// TIA Portal V21 program export: 0 tag tables, 0 data types, 1 data blocks, 5 code blocks (in call order from the OBs), 1 instance data blocks

DATA_BLOCK "Calc"   // DB1
{ S7_Optimized_Access := 'TRUE' }
// stored: MemoryReserve 100
   VAR
      reale : Array[0..100] of LReal;
      tempociclo : LReal;
      tempociclo_T : LReal;
      interi : Array[0..10] of Int;
      tempo : LReal;
      pulse : Array[0..30] of Bool;
   END_VAR
BEGIN
END_DATA_BLOCK

ORGANIZATION_BLOCK "Main"   // OB1, LAD, ProgramCycle
TITLE = "Main Program Sweep (Cycle)"
{ S7_Optimized_Access := 'TRUE' }
// stored: SetENOAutomatically false
   VAR_INPUT
      Initial_Call : Bool;
      Remanence : Bool;
   END_VAR
   VAR_TEMP
      virposINT : DInt;
   END_VAR
BEGIN
END_ORGANIZATION_BLOCK

ORGANIZATION_BLOCK "Cyclic interrupt"   // OB30, LAD, CyclicInterrupt
{ S7_Optimized_Access := 'TRUE' }
// stored: CyclicTime 5000, SetENOAutomatically false
   VAR_INPUT
      Initial_Call : Bool;
      Event_Count : Int;
   END_VAR
   VAR_TEMP
      virposINT : DInt;
      appo : Real;
      VirOnTarget : Bool;
   END_VAR
   VAR_TEMP   // added for the SCL form of the ladder/FBD networks
      _w1 : Bool;
      _w2 : Bool;
      _w3 : Bool;
      _w4 : Bool;
      _w5 : Bool;
      _w6 : Bool;
   END_VAR
BEGIN

REGION Network 2
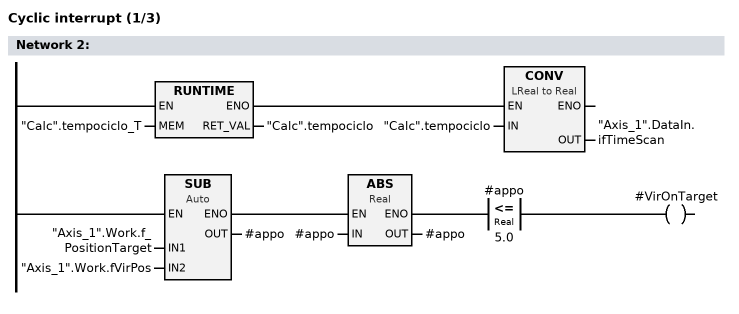
   // no SCL statement known for Runtime: written as a call
   // ENO of a box is taken as its EN; it also drops when the box reports an error
   "Calc".tempociclo := Runtime(mem := "Calc".tempociclo_T);
   "Axis_1".DataIn.ifTimeScan := LREAL_TO_REAL("Calc".tempociclo);
   #appo := "Axis_1".Work.f_PositionTarget - "Axis_1".Work.fVirPos;
   #appo := ABS(#appo);
   #VirOnTarget := #appo <= 5.0;
END_REGION

REGION Network 3
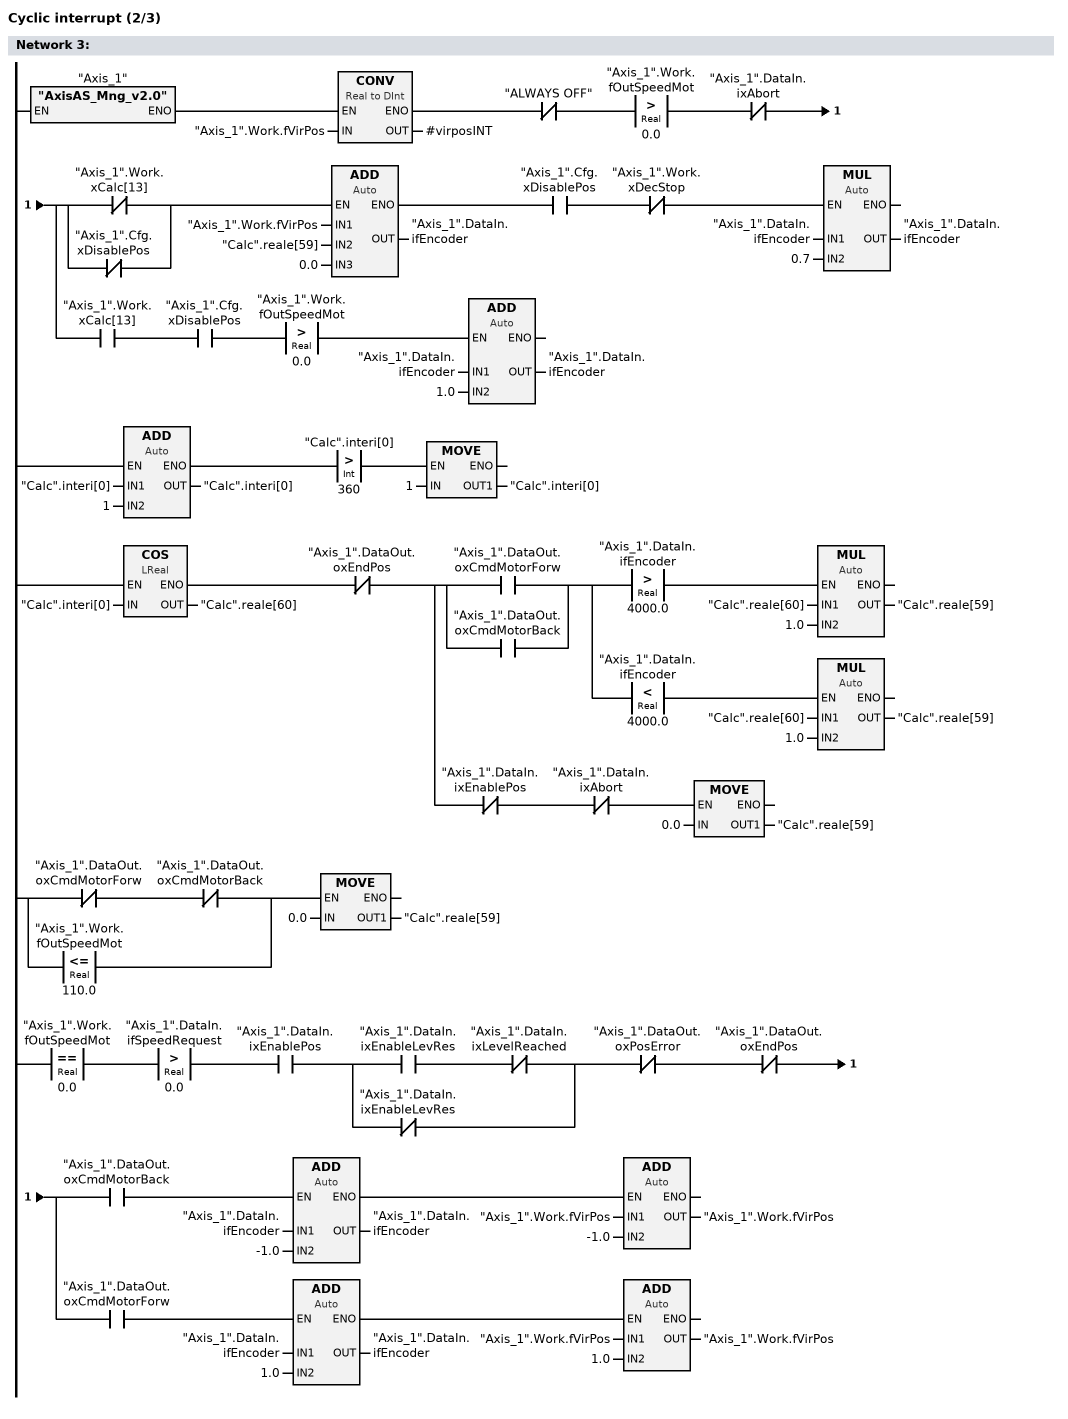
   "Axis_1"(ENO => #_w1);   // "AxisAS_Mng_v2.0"
   IF #_w1 THEN #virposINT := REAL_TO_DINT("Axis_1".Work.fVirPos); END_IF;
   #_w2 := #_w1 AND NOT "ALWAYS OFF" AND ("Axis_1".Work.fOutSpeedMot > 0.0) AND NOT "Axis_1".DataIn.ixAbort;
   #_w3 := #_w2 AND (NOT "Axis_1".Work.xCalc[13] OR NOT "Axis_1".Cfg.xDisablePos);
   IF #_w3 THEN "Axis_1".DataIn.ifEncoder := "Axis_1".Work.fVirPos + "Calc".reale[59] + 0.0; END_IF;
   IF #_w3 AND "Axis_1".Cfg.xDisablePos AND NOT "Axis_1".Work.xDecStop THEN
       "Axis_1".DataIn.ifEncoder := "Axis_1".DataIn.ifEncoder * 0.7;
   END_IF;
   IF #_w2 AND "Axis_1".Work.xCalc[13] AND "Axis_1".Cfg.xDisablePos AND ("Axis_1".Work.fOutSpeedMot > 0.0) THEN
       "Axis_1".DataIn.ifEncoder := "Axis_1".DataIn.ifEncoder + 1.0;
   END_IF;
   "Calc".interi[0] := "Calc".interi[0] + 1;
   IF "Calc".interi[0] > 360 THEN "Calc".interi[0] := 1; END_IF;
   "Calc".reale[60] := COS("Calc".interi[0]);
   #_w4 := NOT "Axis_1".DataOut.oxEndPos;
   #_w5 := #_w4 AND ("Axis_1".DataOut.oxCmdMotorForw OR "Axis_1".DataOut.oxCmdMotorBack);
   IF #_w5 AND ("Axis_1".DataIn.ifEncoder > 4000.0) THEN "Calc".reale[59] := "Calc".reale[60] * 1.0; END_IF;
   IF #_w5 AND ("Axis_1".DataIn.ifEncoder < 4000.0) THEN "Calc".reale[59] := "Calc".reale[60] * 1.0; END_IF;
   IF #_w4 AND NOT "Axis_1".DataIn.ixEnablePos AND NOT "Axis_1".DataIn.ixAbort THEN
       "Calc".reale[59] := 0.0;
   END_IF;
   IF (NOT "Axis_1".DataOut.oxCmdMotorForw AND NOT "Axis_1".DataOut.oxCmdMotorBack) OR ("Axis_1".Work.fOutSpeedMot <= 110.0) THEN
       "Calc".reale[59] := 0.0;
   END_IF;
   #_w6 := ("Axis_1".Work.fOutSpeedMot = 0.0) AND ("Axis_1".DataIn.ifSpeedRequest > 0.0) AND "Axis_1".DataIn.ixEnablePos AND (("Axis_1".DataIn.ixEnableLevRes AND NOT "Axis_1".DataIn.ixLevelReached) OR NOT "Axis_1".DataIn.ixEnableLevRes) AND NOT "Axis_1".DataOut.oxPosError AND NOT "Axis_1".DataOut.oxEndPos;
   IF #_w6 AND "Axis_1".DataOut.oxCmdMotorBack THEN
       "Axis_1".DataIn.ifEncoder := "Axis_1".DataIn.ifEncoder + (-1.0);
       "Axis_1".Work.fVirPos := "Axis_1".Work.fVirPos + (-1.0);
   END_IF;
   IF #_w6 AND "Axis_1".DataOut.oxCmdMotorForw THEN
       "Axis_1".DataIn.ifEncoder := "Axis_1".DataIn.ifEncoder + 1.0;
       "Axis_1".Work.fVirPos := "Axis_1".Work.fVirPos + 1.0;
   END_IF;
END_REGION

REGION Network 4
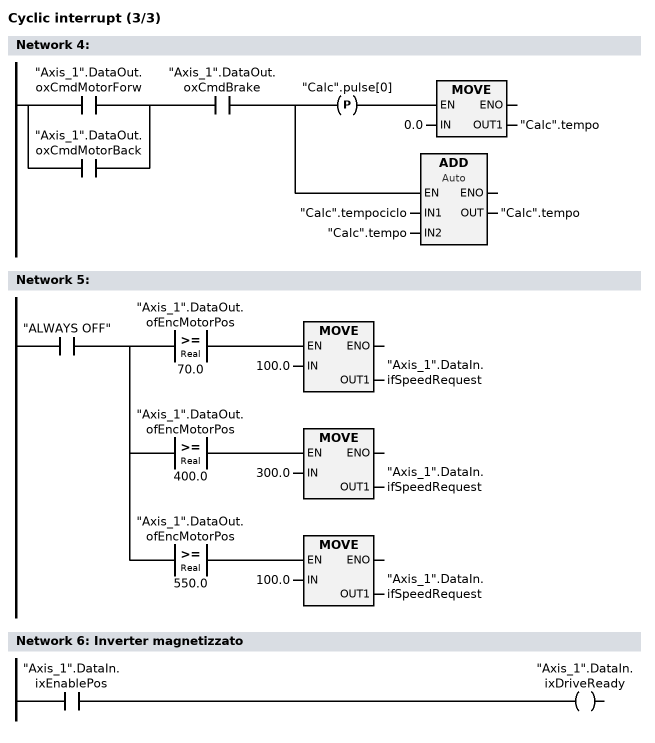
   RUNG wire#powerrail
      Contact( "Axis_1".DataOut.oxCmdMotorForw )
      wire#w1
      Contact( "Axis_1".DataOut.oxCmdBrake )
      wire#w2
      P_Trig( "Calc".pulse[0] )
      Move(in := 0.0, out1 => "Calc".tempo)
   END_RUNG
   RUNG wire#powerrail
      Contact( "Axis_1".DataOut.oxCmdMotorBack )
   END_RUNG wire#w1
   RUNG wire#w2
      Add(in1 := "Calc".tempociclo, in2 := "Calc".tempo, out => "Calc".tempo)
   END_RUNG
   // the same network as SCL:
   #_w1 := ("Axis_1".DataOut.oxCmdMotorForw OR "Axis_1".DataOut.oxCmdMotorBack) AND "Axis_1".DataOut.oxCmdBrake;
   #_w2 := #_w1 AND NOT "Calc".pulse[0];   // rising edge
   "Calc".pulse[0] := #_w1;
   IF #_w2 THEN "Calc".tempo := 0.0; END_IF;
   IF #_w1 THEN "Calc".tempo := "Calc".tempociclo + "Calc".tempo; END_IF;
END_REGION

REGION Network 5
   RUNG wire#powerrail
      Contact( "ALWAYS OFF" )
      wire#w1
      { S7_Templates := "SrcType := Real" } GE_Contact(in1 := "Axis_1".DataOut.ofEncMotorPos, in2 := 70.0)
      Move(in := 100.0, out1 => "Axis_1".DataIn.ifSpeedRequest)
   END_RUNG
   RUNG wire#w1
      { S7_Templates := "SrcType := Real" } GE_Contact(in1 := "Axis_1".DataOut.ofEncMotorPos, in2 := 400.0)
      Move(in := 300.0, out1 => "Axis_1".DataIn.ifSpeedRequest)
   END_RUNG
   RUNG wire#w1
      { S7_Templates := "SrcType := Real" } GE_Contact(in1 := "Axis_1".DataOut.ofEncMotorPos, in2 := 550.0)
      Move(in := 100.0, out1 => "Axis_1".DataIn.ifSpeedRequest)
   END_RUNG
   // the same network as SCL:
   IF "ALWAYS OFF" AND ("Axis_1".DataOut.ofEncMotorPos >= 70.0) THEN
       "Axis_1".DataIn.ifSpeedRequest := 100.0;
   END_IF;
   IF "ALWAYS OFF" AND ("Axis_1".DataOut.ofEncMotorPos >= 400.0) THEN
       "Axis_1".DataIn.ifSpeedRequest := 300.0;
   END_IF;
   IF "ALWAYS OFF" AND ("Axis_1".DataOut.ofEncMotorPos >= 550.0) THEN
       "Axis_1".DataIn.ifSpeedRequest := 100.0;
   END_IF;
END_REGION

REGION Network 6: Inverter magnetizzato
   RUNG wire#powerrail
      Contact( "Axis_1".DataIn.ixEnablePos )
      Coil( "Axis_1".DataIn.ixDriveReady )
   END_RUNG
   // the same network as SCL:
   "Axis_1".DataIn.ixDriveReady := "Axis_1".DataIn.ixEnablePos;
END_REGION
END_ORGANIZATION_BLOCK

FUNCTION_BLOCK "AxisAS_Mng_v2.0"   // FB83, LAD
TITLE = Controllo asse v2.0
{ S7_Optimized_Access := 'TRUE' }
VERSION : 1.0
// stored: MemoryReserve 100, SetENOAutomatically false
   VAR RETAIN
      DataIn : "AxixAS_DataIn_Type_v2.0";
      DataOut : "AxixAS_DataOut_Type_v2.0";
   END_VAR
   VAR
      Sincro { S7_SetPoint := 'True'} : "AxixAS_DataSincro_Type_v2.0";
   END_VAR
   VAR RETAIN
      Cfg { S7_SetPoint := 'True'} : "AxixAS_CFG_Type_v2.0";   // Configurazione Asse
      Work : Struct   // Gestione Asse
         xEnablePos { S7_SetPoint := 'True'} : Bool;   // Posizionatore abilitato/Positioner enabled
         xINEnable : Bool;   // Memo Posizionatore abilitato per inversione
         xDriveReady { S7_SetPoint := 'True'} : Bool;   // Inverter magnetizzato
         xCmdVirSpeedChanged { S7_SetPoint := 'True'} : Bool;   // Variazione target VEL durante missione
         "xCurveS-L" { ExternalWritable := 'False'; S7_SetPoint := 'True'} : Bool;   // Curva non lineare
         "xAutoChangeS-L" { S7_SetPoint := 'True'} : Bool;   // Autoimpostazione LIN per brevi spostamenti
         "xCTRAutoChangeS-L" { S7_SetPoint := 'True'} : Bool;   // Autoimpostazione LIN per brevi spostamenti
         xDecStop { S7_SetPoint := 'True'} : Bool;   // Inizio dec. per raggiungimento quota richiesta
         xDecResearch { S7_SetPoint := 'True'} : Bool;   // Inizio decelerazione per passaggio a velocità ricerca livello
         xStopVirPositioner { S7_SetPoint := 'True'} : Bool;   // Arresto posizionatore Target raggiunto
         xEnableJog { S7_SetPoint := 'True'} : Bool;   // JOG movimento in corso
         xChangeTargetPulse { S7_SetPoint := 'True'} : Bool;   // Target changed
         xAutoSpeedPulse { S7_SetPoint := 'True'} : Bool;   // Enable AutoSpeed pulse
         xEnablePulse { S7_SetPoint := 'True'} : Bool;   // Enable pulse
         f_PositionTarget { S7_SetPoint := 'True'} : Real;   // Posizione Richiesta Target
         fVirPos { S7_SetPoint := 'True'} : Real;   // Posizione encoder Asse virtuale (mm)
         f_SpeedReqCalc { S7_SetPoint := 'True'} : Real;   // Velocità TARGET autocalcolata su spazio destinazione
         fVirSpeed { S7_SetPoint := 'True'} : Real;   // Velocità Asse virtuale (mm/sec) TRA-LOG-COS
         fVirSpeedLinear { S7_SetPoint := 'True'} : Real;   // Velocità Asse LINEARE
         fVirSpeedLog { S7_SetPoint := 'True'} : Real;   // Velocità Asse LOGARITMICA
         fVirSpeedCos { S7_SetPoint := 'True'} : Real;   // Velocità Asse COSENO
         fCmdVirSpeed { S7_SetPoint := 'True'} : Real;   // Velocità richiesta Asse (mm/sec)
         fCmdVirSpeedMemo { S7_SetPoint := 'True'} : Real;   // Memo Velocità richiesta Asse (mm/sec)
         fCmdVirAcc { S7_SetPoint := 'True'} : Real;   // Acc. richiesta Asse (mm/sec^2)
         fCmdVirDec { S7_SetPoint := 'True'} : Real;   // Dec. richiesta Asse (mm/sec^2)
         fLimVirDec { S7_SetPoint := 'True'} : Real;   // * Limite massimo dec. modulata per fermata
         fDecVirStop { S7_SetPoint := 'True'} : Real;   // * Dec. richiesta per posizionatore stop quota (mm/sec^2)
         fCalcEncErr { S7_SetPoint := 'True'} : Real;   // * Errore tra pos. attuale e reale encoder motore
         fJogSpeed { S7_SetPoint := 'True'} : Real;   // Velocità JOG (mm/sec)
         fCmdJogSpeed { S7_SetPoint := 'True'} : Real;   // Velocità richiesta JOG (mm/sec)
         fCmdJogAcc { S7_SetPoint := 'True'} : Real;   // Acc. richiesta JOG (mm/sec^2)
         fCmdJogDec { S7_SetPoint := 'True'} : Real;   // Dec. richiesta JOG (mm/sec^2)
         "fLim+Ppid" { S7_SetPoint := 'True'} : Real;   // Limite massimo positivo azione proporzionale (20% velocità massima)
         "fLim-Ppid" { S7_SetPoint := 'True'} : Real;   // Limite massimo negativo azione proporzionale (20% velocità massima)
         fOutSpeedMot { S7_SetPoint := 'True'} : Real;   // Velocità comando motore da POS o JOG
         fSuppCalcPpid { S7_SetPoint := 'True'} : Real;   // App calcolo proporzionale
         fMemoMaxSpeed { S7_SetPoint := 'True'} : Real;   // Memorizzo velocità massima (mm/sec)
         fPpid { S7_SetPoint := 'True'} : Real;   // Parte P del Pid
         fMemoOldPos { S7_SetPoint := 'True'} : Real;   // Quota Old/Position Old (mm)
         fAccOnWork { S7_SetPoint := 'True'} : Real;   // Accelerazione calcolata/imposta
         fDecOnWork { S7_SetPoint := 'True'} : Real;   // Decelerazione calcolata/imposta
         fSpaceFromTarget : Real;   // Spazio autocalcolo memo
         xTimBrakeDelay_Fwd : Bool;   // Ritardo sgancio freno FWD
         xTimBrakeDelay_Bkw : Bool;   // Ritardo sgancio freno BKW
         xTimStopEndPos : Bool;   // Ritardo allarme controllo fine posizionamento
         xMotorMagn_pulse : Bool;   // Mem richiesta esterna magnetizzazione DataIn
         fCalc : Array[0..20] of Real;
         xCalc : Array[0..20] of Bool;
      END_STRUCT;
   END_VAR
   VAR
      TmrBrake_Fwd : IEC_TIMER;   // Timer sgancio freno FWD
      TmrBrake_Bkw : IEC_TIMER;   // Timer sgancio freno BKW
      Tmr_EndPos : IEC_TIMER;   // Timer allarme controllo fine posizionamento
      Tmr_DriveOnReq : IEC_TIMER;   // Timer OFF richiesta Drive Ready
      Tmr_DriveOffReq : IEC_TIMER;   // Timer ON richiesta Drive Ready
      Tmr_OnMove : IEC_TIMER;
   END_VAR
   VAR_TEMP
      tfSuppCalc : Real;   // Appoggio per calcoli
      fSlopeAccLog : Real;
      fSlopeDecLog : Real;
      fSlopeAccCos : Real;
      fSlopeDecCos : Real;
      fCalcSpeed : Real;
      fCalcAppo : Real;
      oxCmdMotorFWD : Bool;
      oxCmdMotorBKW : Bool;
      fCalcSpaceOff : Real;
      xDummy : Bool;
      xMotorPulse : Bool;
      y : Real;
      x : Real;
      "m" : Real;
      q : Real;
   END_VAR
   VAR CONSTANT
      PiGrego : Real := 3.141593;
      "100Sec" : Time := T#100s;
   END_VAR
   VAR_TEMP   // added for the SCL form of the ladder/FBD networks
      _w1 : Bool;
      _w2 : Bool;
      _w3 : Bool;
   END_VAR
BEGIN

REGION Network 1 (SCL): Descrizione funzionamento e Versioni
   (*
   ------------------------------------------------------------------------
   AUTHOR:     M.Montanari
   DATE:       06/06/2022
   VERSION:    v0.0
   ------------------------------------------------------------------------

   DESCRIPTION: "AxisAs_Mng"
       Gestore ASSE per motore asincrono con posizionatore a generazione di profilo ed inseguimento proporzionale + piramidale

       Implements the following functions:

   WORKING: (funzionamento)

   - Curva Trapezio
   - Curva "esse" logaritmica
   - Auto gestione curva per piccoli spostamenti
   - Attesa segnale inverter magnetizzato

   INPUT:

   OUTPUT:

   INOUT:

   DEPENDENCIES: (dipendenze: FB, FC, DataTypes, etc...)
       ...

   USAGE (utilizzo):

   NOTES:
      il buon funzionamento del sistema dipende anche dalla parametrizzazione dell'inverter.
      di seguito alcuni parametri da sistemare se si utilizzano Inverters Siemens.

   - Wizard impostare generazione RAMPE NEL PLC
   - Tipo di regolazione p1300 = [1] Controllo U/f con caretteristica lineare e FCC
   - Parametrizzare freno p1215 =[3] freno staz mot come contr. sew. colleg. tramite BICO 
   - tempi p1216=50ms p1217=40ms
   - p1120[0] Tempo di accelerazione del generatore di rampa --> 0,00s
   - p1121[0] Tempo di decelerazione del generatore di rampa --> 0,00s
   - p1127[0] Generatore di rampa, tempo di decelerazione minimo --> 0,154s
   - Tempo OFF3 p1135=0,020s
   - Limite di corrente 2 volte corrente nominale motore
   - Non toccare tempi magnetizzazione/demagnetizzazione calcolati
   - Fare autotuning per carichi sospesi o sbilanciati
   - Boost p1310=50% p1311=25% p1312=0%


   ------------------------------------------------------------------------
   TODO:
      ...

   CHANGELOG:

   v2.0 - 01/03/2024 - Michele Montanari
       - Aggiornamento struttura CFG, DataIn, Sincro : 
           - inserita configurazione retta di adeguamento autospeed
           - inserito soglia Acc/Dec minima su autocalcolo e soglia intervento autospeed
           - inserito modalità che disabilita il controllo asse e rende il controllo in anello aperto
           - ricerca livello con TRIGGER esterno, stop moto gestito autonomamente
           - ricerca livello in entrambi i sensi di moto
           - aggiornamento continuo ctr valori anello posizione di VirSpeed
           - predisposizione funzione assi Geraing & Sincro
   ------------------------------------------------------------------------
   *)
END_REGION

REGION Network 2 (SCL): Autocalcolo velocità su spazio da percorrere
   IF NOT #DataIn.xAutoSpeedDetect THEN
       #Work.f_SpeedReqCalc := #DataIn.ifSpeedRequest;
   END_IF;

   IF #DataOut.ofSpeedRequest > 0 AND #Work.fVirSpeed > 0 THEN
       #Work.xAutoSpeedPulse := FALSE;
   END_IF;

   IF #DataIn.xAutoSpeedDetect AND (ABS(#DataIn.ifPositionRequest - #DataIn.ifEncoder) <= #Cfg.fThreshold_SUP_AutoSpeed) THEN
       IF #DataOut.ofSpeedRequest = 0 AND #Work.fVirSpeed = 0 THEN //AND NOT #Work.xEnablePulse THEN
           #Work.xAutoSpeedPulse := TRUE;
           #Work.fSpaceFromTarget := ABS(#DataIn.ifPositionRequest - #DataIn.ifEncoder);

           #x := #Work.fSpaceFromTarget;
           IF #x < #Cfg.fThreshold_INF_AutoSpeed THEN
               #x := #Cfg.fThreshold_INF_AutoSpeed;
           END_IF;
           #m := (#Cfg.fMaxSpeed - #Cfg.fMinSpeed) / (#Cfg.fThreshold_SUP_AutoSpeed - #Cfg.fThreshold_INF_AutoSpeed);
           #q := #Cfg.fMinSpeed - #m * #Cfg.fThreshold_INF_AutoSpeed;
           #y := #m * #x + #q;

           #fCalcSpeed := ABS(#y);

           IF #fCalcSpeed > #DataIn.ifSpeedRequest THEN
               #Work.f_SpeedReqCalc := #DataIn.ifSpeedRequest;
           ELSE
               #Work.f_SpeedReqCalc := #fCalcSpeed;
           END_IF;
       END_IF;

       ELSE

           #Work.f_SpeedReqCalc := #DataIn.ifSpeedRequest;
    END_IF;



   IF #Work.f_SpeedReqCalc > #Cfg.fMaxSpeed THEN
       #Work.f_SpeedReqCalc := #Cfg.fMaxSpeed;
   END_IF;
END_REGION

REGION Network 3: Accetta nuova destinazione se fermo o oltre target e si arresta subito per fare inversione se prima del target
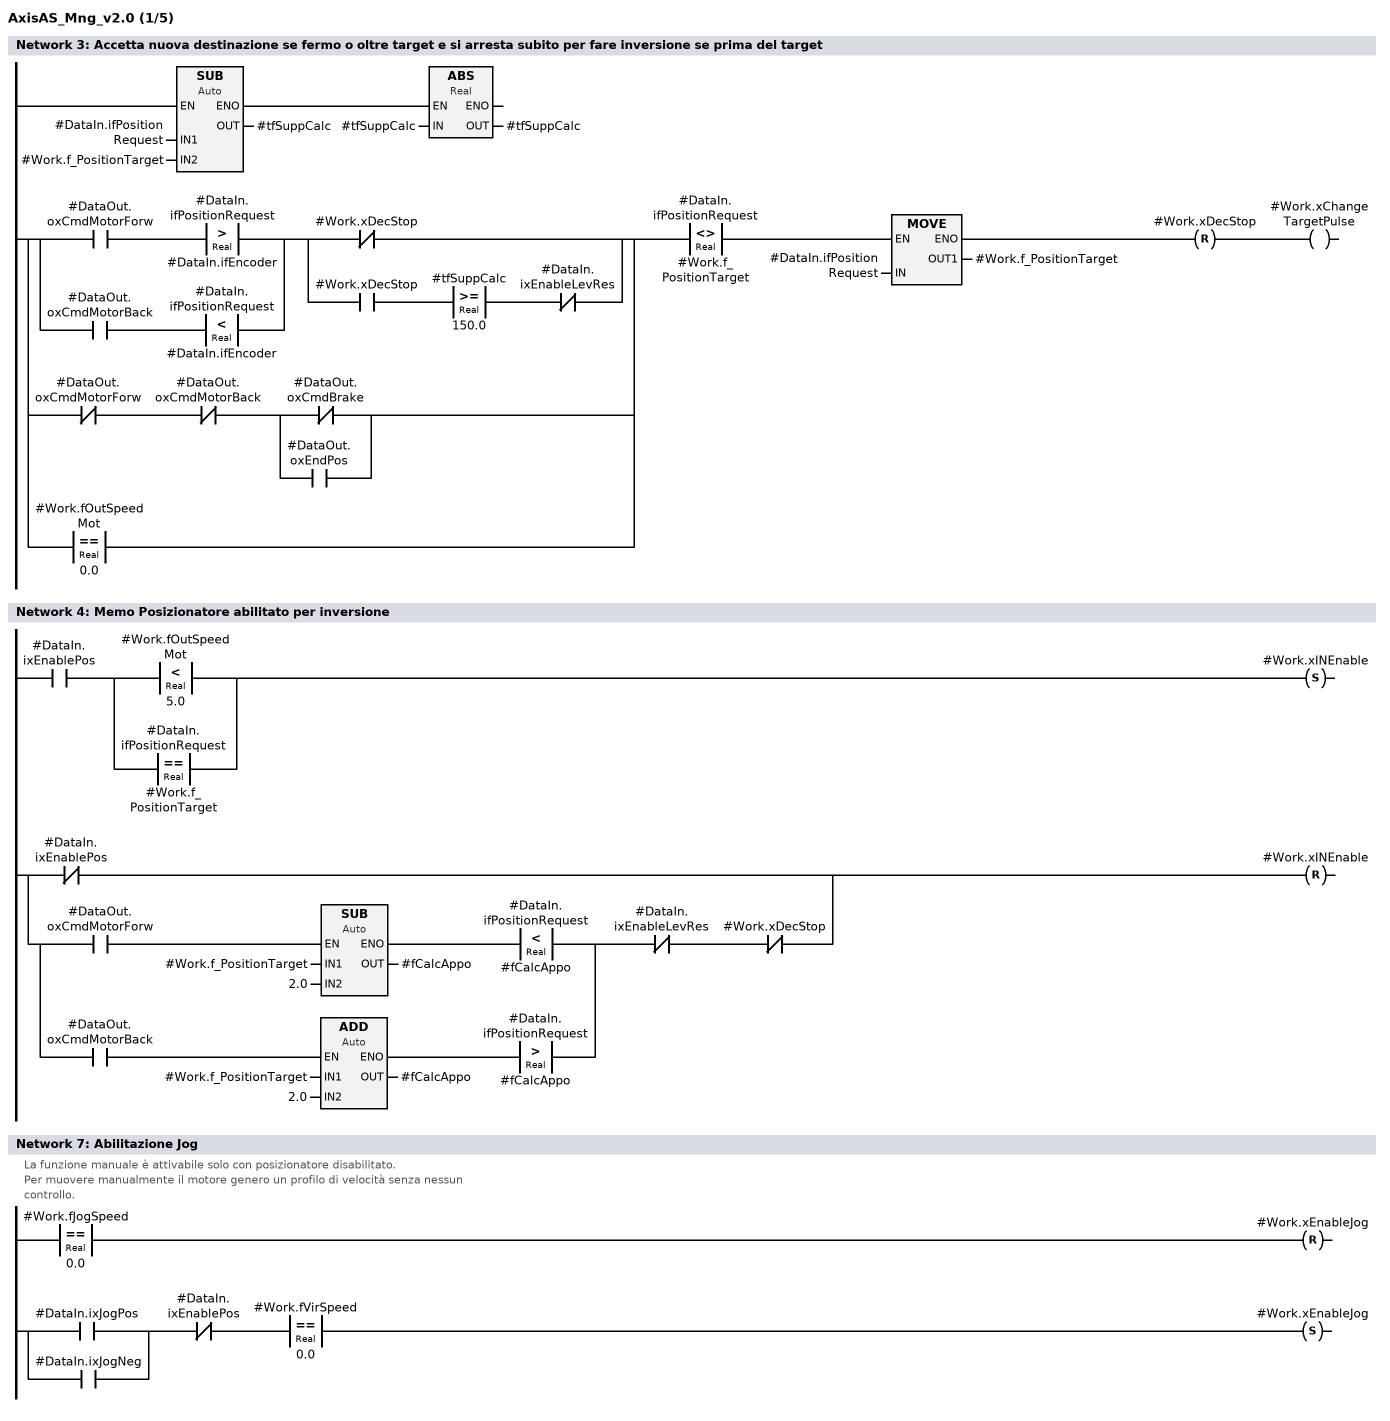
   RUNG wire#powerrail
      Sub(in1 := #DataIn.ifPositionRequest, in2 := #Work.f_PositionTarget, out => #tfSuppCalc)
      { S7_Templates := "SrcType := Real" } Abs(in := #tfSuppCalc, out => #tfSuppCalc)
   END_RUNG
   RUNG wire#powerrail
      Contact( #DataOut.oxCmdMotorForw )
      { S7_Templates := "SrcType := Real" } GT_Contact(in1 := #DataIn.ifPositionRequest, in2 := #DataIn.ifEncoder)
      wire#w1
      I_Contact( #Work.xDecStop )
      wire#w2
      { S7_Templates := "SrcType := Real" } NE_Contact(in1 := #DataIn.ifPositionRequest, in2 := #Work.f_PositionTarget)
      Move(in := #DataIn.ifPositionRequest, out1 => #Work.f_PositionTarget)
      R_Coil( #Work.xDecStop )
      Coil( #Work.xChangeTargetPulse )
   END_RUNG
   RUNG wire#powerrail
      Contact( #DataOut.oxCmdMotorBack )
      { S7_Templates := "SrcType := Real" } LT_Contact(in1 := #DataIn.ifPositionRequest, in2 := #DataIn.ifEncoder)
   END_RUNG wire#w1
   RUNG wire#w1
      Contact( #Work.xDecStop )
      { S7_Templates := "SrcType := Real" } GE_Contact(in1 := #tfSuppCalc, in2 := 150.0)
      I_Contact( #DataIn.ixEnableLevRes )
   END_RUNG wire#w2
   RUNG wire#powerrail
      I_Contact( #DataOut.oxCmdMotorForw )
      I_Contact( #DataOut.oxCmdMotorBack )
      wire#w3
      I_Contact( #DataOut.oxCmdBrake )
   END_RUNG wire#w2
   RUNG wire#w3
      Contact( #DataOut.oxEndPos )
   END_RUNG wire#w2
   RUNG wire#powerrail
      { S7_Templates := "SrcType := Real" } EQ_Contact(in1 := #Work.fOutSpeedMot, in2 := 0.0)
   END_RUNG wire#w2
   // the same network as SCL:
   #tfSuppCalc := #DataIn.ifPositionRequest - #Work.f_PositionTarget;
   #tfSuppCalc := ABS(#tfSuppCalc);
   #_w1 := ((((#DataOut.oxCmdMotorForw AND (#DataIn.ifPositionRequest > #DataIn.ifEncoder)) OR (#DataOut.oxCmdMotorBack AND (#DataIn.ifPositionRequest < #DataIn.ifEncoder))) AND (NOT #Work.xDecStop OR (#Work.xDecStop AND (#tfSuppCalc >= 150.0) AND NOT #DataIn.ixEnableLevRes))) OR (NOT #DataOut.oxCmdMotorForw AND NOT #DataOut.oxCmdMotorBack AND (NOT #DataOut.oxCmdBrake OR #DataOut.oxEndPos)) OR (#Work.fOutSpeedMot = 0.0)) AND (#DataIn.ifPositionRequest <> #Work.f_PositionTarget);
   IF #_w1 THEN
       #Work.f_PositionTarget := #DataIn.ifPositionRequest;
       #Work.xDecStop := FALSE;
   END_IF;
   #Work.xChangeTargetPulse := #_w1;
END_REGION

REGION Network 4: Memo Posizionatore abilitato per inversione
   RUNG wire#powerrail
      Contact( #DataIn.ixEnablePos )
      wire#w1
      { S7_Templates := "SrcType := Real" } LT_Contact(in1 := #Work.fOutSpeedMot, in2 := 5.0)
      wire#w2
      S_Coil( #Work.xINEnable )
   END_RUNG
   RUNG wire#w1
      { S7_Templates := "SrcType := Real" } EQ_Contact(in1 := #DataIn.ifPositionRequest, in2 := #Work.f_PositionTarget)
   END_RUNG wire#w2
   RUNG wire#powerrail
      I_Contact( #DataIn.ixEnablePos )
      wire#w3
      R_Coil( #Work.xINEnable )
   END_RUNG
   RUNG wire#powerrail
      Contact( #DataOut.oxCmdMotorForw )
      Sub(in1 := #Work.f_PositionTarget, in2 := 2.0, out => #fCalcAppo)
      { S7_Templates := "SrcType := Real" } LT_Contact(in1 := #DataIn.ifPositionRequest, in2 := #fCalcAppo)
      wire#w4
      I_Contact( #DataIn.ixEnableLevRes )
      I_Contact( #Work.xDecStop )
   END_RUNG wire#w3
   RUNG wire#powerrail
      Contact( #DataOut.oxCmdMotorBack )
      Add(in1 := #Work.f_PositionTarget, in2 := 2.0, out => #fCalcAppo)
      { S7_Templates := "SrcType := Real" } GT_Contact(in1 := #DataIn.ifPositionRequest, in2 := #fCalcAppo)
   END_RUNG wire#w4
   // the same network as SCL:
   IF #DataIn.ixEnablePos AND ((#Work.fOutSpeedMot < 5.0) OR (#DataIn.ifPositionRequest = #Work.f_PositionTarget)) THEN
       #Work.xINEnable := TRUE;
   END_IF;
   IF #DataOut.oxCmdMotorForw THEN #fCalcAppo := #Work.f_PositionTarget - 2.0; END_IF;
   #_w1 := #DataOut.oxCmdMotorForw AND (#DataIn.ifPositionRequest < #fCalcAppo);
   IF #DataOut.oxCmdMotorBack THEN #fCalcAppo := #Work.f_PositionTarget + 2.0; END_IF;
   IF NOT #DataIn.ixEnablePos OR ((#_w1 OR (#DataOut.oxCmdMotorBack AND (#DataIn.ifPositionRequest > #fCalcAppo))) AND NOT #DataIn.ixEnableLevRes AND NOT #Work.xDecStop) THEN
       #Work.xINEnable := FALSE;
   END_IF;
END_REGION

REGION Network 5 (SCL): Autocalcolo ACC-DEC su velocità
   IF #DataIn.xAutoAccDecCalculation THEN
       #Work.fAccOnWork := #Cfg.fMaxAccRamp * (#Work.f_SpeedReqCalc / #Cfg.fMaxSpeed);
       #Work.fDecOnWork := #Cfg.fMaxDecRamp * (#Work.f_SpeedReqCalc / #Cfg.fMaxSpeed);
   ELSE
       #Work.fAccOnWork := #DataIn.ifAccRamp;
       #Work.fDecOnWork := #DataIn.ifDecRamp;
   END_IF;

   IF #Work.fAccOnWork < #Cfg.fMinAccRamp THEN
       #Work.fAccOnWork := #Cfg.fMinAccRamp;
   END_IF;
   IF #Work.fDecOnWork < #Cfg.fMinDecRamp THEN
       #Work.fDecOnWork := #Cfg.fMinDecRamp;
   END_IF;
   IF #Work.fAccOnWork > #Cfg.fMaxAccRamp THEN
       #Work.fAccOnWork := #Cfg.fMaxAccRamp;
   END_IF;
   IF #Work.fDecOnWork > #Cfg.fMaxDecRamp THEN
       #Work.fDecOnWork := #Cfg.fMaxDecRamp;
   END_IF;
END_REGION

REGION Network 6 (SCL): Selezione curva
   // Per spostamenti inferiori a  #CFG."fAutoChangeS-Lvalue" impone una curva a TRA se selezionata LOG
   CASE #Cfg."xCurveS-L" OF
       0:  // Statement section case 1
           #Work."xCurveS-L" := FALSE;
       1:  // Statement section case 2 to 4
           IF (#Work.xINEnable) AND NOT #Work."xCTRAutoChangeS-L" THEN
               #Work."xCTRAutoChangeS-L" := TRUE;
               IF (ABS(#Work.f_PositionTarget - #DataIn.ifEncoder) < #Cfg."fAutoChangeS-Lvalue") THEN
                   #Work."xAutoChangeS-L" := TRUE;
               END_IF;
           END_IF;
           IF #Work."xAutoChangeS-L" THEN
               #Work."xCurveS-L" := FALSE;
           ELSE
               #Work."xCurveS-L" := TRUE;
           END_IF;
       2:  // Statement section case 2 to 4
           #Work."xCurveS-L" := TRUE;
   END_CASE;

   IF NOT #Work.xINEnable AND NOT #Work.xDecStop THEN
       #Work."xCTRAutoChangeS-L" := FALSE;
   END_IF;
   IF ABS(#Work.f_PositionTarget -  #DataIn.ifEncoder) <= #Cfg.fVirt_EncWindPos THEN
       #Work."xAutoChangeS-L" := FALSE;
   END_IF;
END_REGION

REGION Network 7: Abilitazione Jog
   // La funzione manuale è attivabile solo con posizionatore disabilitato.
   // Per muovere manualmente il motore genero un profilo di velocità senza nessun 
   // controllo.
   RUNG wire#powerrail
      { S7_Templates := "SrcType := Real" } EQ_Contact(in1 := #Work.fJogSpeed, in2 := 0.0)
      R_Coil( #Work.xEnableJog )
   END_RUNG
   RUNG wire#powerrail
      Contact( #DataIn.ixJogPos )
      wire#w1
      I_Contact( #DataIn.ixEnablePos )
      { S7_Templates := "SrcType := Real" } EQ_Contact(in1 := #Work.fVirSpeed, in2 := 0.0)
      S_Coil( #Work.xEnableJog )
   END_RUNG
   RUNG wire#powerrail
      Contact( #DataIn.ixJogNeg )
   END_RUNG wire#w1
   // the same network as SCL:
   IF #Work.fJogSpeed = 0.0 THEN #Work.xEnableJog := FALSE; END_IF;
   IF (#DataIn.ixJogPos OR #DataIn.ixJogNeg) AND NOT #DataIn.ixEnablePos AND (#Work.fVirSpeed = 0.0) THEN
       #Work.xEnableJog := TRUE;
   END_IF;
END_REGION

REGION Network 8 (SCL): Attivazione funzionamento di jog
   // Con abilitazione attiva carico velocità jog e inizio generazione profilo di velocità senza alcun controllo
   IF #Work.xEnableJog THEN

       IF #DataIn.ixJogPos OR #DataIn.ixJogNeg THEN
           #Work.fCmdJogSpeed := #Cfg.fJogSpeed;
       ELSE
           #Work.fCmdJogSpeed := 0.0;
       END_IF;

       IF #Work.fJogSpeed >= 0.0 THEN
           #Work.fCmdJogAcc := #Cfg.fJogAcc * #DataIn.ifTimeScan;
           #Work.fCmdJogDec := #Cfg.fJogDec * #DataIn.ifTimeScan;
       END_IF;

       IF #Work.fCmdJogSpeed > #Work.fJogSpeed THEN
           #Work.fJogSpeed := #Work.fJogSpeed + #Work.fCmdJogAcc;
           IF #Work.fJogSpeed > #Work.fCmdJogSpeed THEN
               #Work.fJogSpeed := #Work.fCmdJogSpeed;
           END_IF;
       END_IF;

       IF #Work.fCmdJogSpeed < #Work.fJogSpeed THEN
           #Work.fJogSpeed := #Work.fJogSpeed - #Work.fCmdJogDec;
           IF #Work.fJogSpeed < #Work.fCmdJogSpeed THEN
               #Work.fJogSpeed := #Work.fCmdJogSpeed;
           END_IF;
       END_IF;

   END_IF;
END_REGION

REGION Network 9: Controllo se posizionatore abilitato e inverter ready
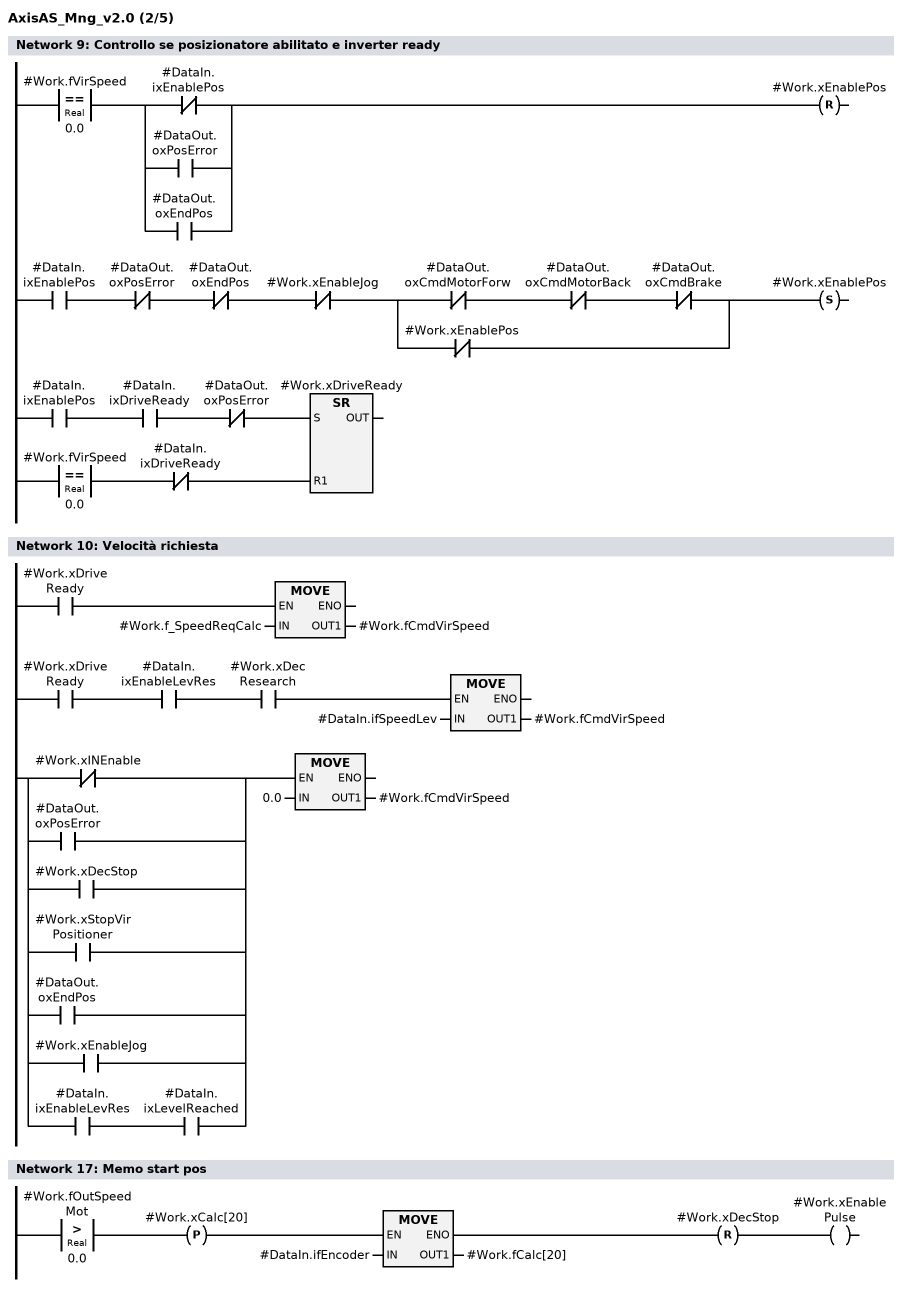
   RUNG wire#powerrail
      { S7_Templates := "SrcType := Real" } EQ_Contact(in1 := #Work.fVirSpeed, in2 := 0.0)
      wire#w1
      I_Contact( #DataIn.ixEnablePos )
      wire#w2
      R_Coil( #Work.xEnablePos )
   END_RUNG
   RUNG wire#w1
      Contact( #DataOut.oxPosError )
   END_RUNG wire#w2
   RUNG wire#w1
      Contact( #DataOut.oxEndPos )
   END_RUNG wire#w2
   RUNG wire#powerrail
      Contact( #DataIn.ixEnablePos )
      I_Contact( #DataOut.oxPosError )
      I_Contact( #DataOut.oxEndPos )
      I_Contact( #Work.xEnableJog )
      wire#w3
      I_Contact( #DataOut.oxCmdMotorForw )
      I_Contact( #DataOut.oxCmdMotorBack )
      I_Contact( #DataOut.oxCmdBrake )
      wire#w4
      S_Coil( #Work.xEnablePos )
   END_RUNG
   RUNG wire#w3
      I_Contact( #Work.xEnablePos )
   END_RUNG wire#w4
   RUNG wire#powerrail
      Contact( #DataIn.ixEnablePos )
      Contact( #DataIn.ixDriveReady )
      I_Contact( #DataOut.oxPosError )
      S_SR(operand := #Work.xDriveReady, r1 := wire#w5)
   END_RUNG
   RUNG wire#powerrail
      { S7_Templates := "SrcType := Real" } EQ_Contact(in1 := #Work.fVirSpeed, in2 := 0.0)
      I_Contact( #DataIn.ixDriveReady )
   END_RUNG wire#w5
   // the same network as SCL:
   IF (#Work.fVirSpeed = 0.0) AND (NOT #DataIn.ixEnablePos OR #DataOut.oxPosError OR #DataOut.oxEndPos) THEN
       #Work.xEnablePos := FALSE;
   END_IF;
   IF #DataIn.ixEnablePos AND NOT #DataOut.oxPosError AND NOT #DataOut.oxEndPos AND NOT #Work.xEnableJog AND ((NOT #DataOut.oxCmdMotorForw AND NOT #DataOut.oxCmdMotorBack AND NOT #DataOut.oxCmdBrake) OR NOT #Work.xEnablePos) THEN
       #Work.xEnablePos := TRUE;
   END_IF;
   IF #DataIn.ixEnablePos AND #DataIn.ixDriveReady AND NOT #DataOut.oxPosError THEN
       #Work.xDriveReady := TRUE;   // SR flip-flop
   END_IF;
   IF (#Work.fVirSpeed = 0.0) AND NOT #DataIn.ixDriveReady THEN #Work.xDriveReady := FALSE; END_IF;
END_REGION

REGION Network 10: Velocità richiesta
   RUNG wire#powerrail
      Contact( #Work.xDriveReady )
      Move(in := #Work.f_SpeedReqCalc, out1 => #Work.fCmdVirSpeed)
   END_RUNG
   RUNG wire#powerrail
      Contact( #Work.xDriveReady )
      Contact( #DataIn.ixEnableLevRes )
      Contact( #Work.xDecResearch )
      Move(in := #DataIn.ifSpeedLev, out1 => #Work.fCmdVirSpeed)
   END_RUNG
   RUNG wire#powerrail
      I_Contact( #Work.xINEnable )
      wire#w1
      Move(in := 0.0, out1 => #Work.fCmdVirSpeed)
   END_RUNG
   RUNG wire#powerrail
      Contact( #DataOut.oxPosError )
   END_RUNG wire#w1
   RUNG wire#powerrail
      Contact( #Work.xDecStop )
   END_RUNG wire#w1
   RUNG wire#powerrail
      Contact( #Work.xStopVirPositioner )
   END_RUNG wire#w1
   RUNG wire#powerrail
      Contact( #DataOut.oxEndPos )
   END_RUNG wire#w1
   RUNG wire#powerrail
      Contact( #Work.xEnableJog )
   END_RUNG wire#w1
   RUNG wire#powerrail
      Contact( #DataIn.ixEnableLevRes )
      Contact( #DataIn.ixLevelReached )
   END_RUNG wire#w1
   // the same network as SCL:
   IF #Work.xDriveReady THEN #Work.fCmdVirSpeed := #Work.f_SpeedReqCalc; END_IF;
   IF #Work.xDriveReady AND #DataIn.ixEnableLevRes AND #Work.xDecResearch THEN
       #Work.fCmdVirSpeed := #DataIn.ifSpeedLev;
   END_IF;
   IF NOT #Work.xINEnable OR #DataOut.oxPosError OR #Work.xDecStop OR #Work.xStopVirPositioner OR #DataOut.oxEndPos OR #Work.xEnableJog OR (#DataIn.ixEnableLevRes AND #DataIn.ixLevelReached) THEN
       #Work.fCmdVirSpeed := 0.0;
   END_IF;
END_REGION

REGION Network 11 (SCL): Calcolo Profilo velocità posizionatore TRAPEZIO

   #Work.fCmdVirAcc := (#Work.fAccOnWork * #DataIn.ifTimeScan);
   #Work.fCmdVirDec := (#Work.fDecOnWork * #DataIn.ifTimeScan);

   IF #Work.fCmdVirSpeed > #Work.fVirSpeedLinear THEN
       #Work.fVirSpeedLinear := #Work.fVirSpeedLinear + #Work.fCmdVirAcc;
       IF #Work.fVirSpeedLinear > #Work.fCmdVirSpeed THEN
           #Work.fVirSpeedLinear := #Work.fCmdVirSpeed;
       END_IF;
   END_IF;

   IF #Work.fCmdVirSpeed <= #Work.fVirSpeedLinear THEN
       #Work.fVirSpeedLinear := #Work.fVirSpeedLinear - #Work.fCmdVirDec;
       IF #Work.fVirSpeedLinear < #Work.fCmdVirSpeed THEN
           #Work.fVirSpeedLinear := #Work.fCmdVirSpeed;
       END_IF;
       IF NOT (#Work.xStopVirPositioner) AND (#Work.fVirSpeedLinear < #Cfg.fMinSpeed)
           AND NOT (#DataOut.oxPosError) AND #Work.xINEnable AND #Work.xDriveReady THEN
           #Work.fVirSpeedLinear := #Cfg.fMinSpeed;
       END_IF;
   END_IF;
END_REGION

REGION Network 12 (SCL): Gestione cambio target velocità log-cos
       IF (#Work.fCmdVirSpeedMemo <> #Work.fCmdVirSpeed) THEN
           IF #Work.fCmdVirSpeed > 0 AND #Work.fCmdVirSpeedMemo <> 0 THEN
               #Work.fCalc[7] := #Work.fVirSpeedLog;
               #Work.fCalc[0] := 0;
               #Work.fCalc[17] := #Work.fVirSpeedCos;
               #Work.fCalc[19] := 0;
               IF #Work.fCmdVirSpeed > #Work.fCmdVirSpeedMemo THEN
                   #Work.xCmdVirSpeedChanged := FALSE;
               ELSE
                   #Work.xCmdVirSpeedChanged := TRUE;
               END_IF;
           END_IF;
           #Work.fCmdVirSpeedMemo := #Work.fCmdVirSpeed;
       END_IF;
END_REGION

REGION Network 13 (SCL): Calcolo Profilo velocità posizionatore LOGARITMICA
   // Calcolo velocità profilo posizionatore.
   // Durante la fase di fermata modulo la decelerazione per fermarmi nella posizione 
   // richiesta; la variazione massima di decelerazione è del 50%. Questo è 
   // necessario in quanto il punto di richiesta velocità 0 è afflitto dall'errore 
   // generato dal tempo di scansione della CPU.

   IF #Work."xCurveS-L" THEN



       IF  #Work.fCalc[10] < #Work.fVirSpeedLog THEN
           #Work.fCalc[10] := #Work.fVirSpeedLog;
       END_IF;
       IF #Work.fVirSpeed = 0 THEN
           #Work.fCalc[10] := 0;
       END_IF;

       IF  #Work.xEnablePulse THEN
           #Work.xCalc[0] := FALSE;
           #Work.fVirSpeed := 0;
           #Work.fCalc[0] := 0;
           #Work.fCalc[4] := 0;
           #Work.fCalc[5] := 0;
           #Work.fCalc[7] := 0;
           #Work.fCalc[10] := 0;
       END_IF;

       #fSlopeAccLog := (12 * #Work.fAccOnWork) / (ABS(#Work.fCmdVirSpeed - #Work.fCalc[7]) + 1);
       #fSlopeDecLog := (12 * #Work.fDecOnWork) / (#Work.fCalc[10] + 1);

       IF #Work.fCmdVirSpeed > 0 THEN
           #Work.fCalc[5] := 1;
           IF #Work.fCalc[5] < #Work.fVirSpeedLog THEN
               #Work.fCalc[5] := #Work.fVirSpeedLog;
           END_IF;
           #Work.fCalc[0] := #Work.fCalc[0] + #DataIn.ifTimeScan;
           IF NOT #Work.xCmdVirSpeedChanged THEN
               #Work.fVirSpeedLog := #Work.fCalc[7] + (#Work.fCmdVirSpeed - #Work.fCalc[7]) * (1 / (1 + EXP(- (#Work.fCalc[0] * #fSlopeAccLog - #Cfg.fFirstStepNepero))));
           ELSE
               #fSlopeDecLog := (12 * #Work.fDecOnWork) / ABS((#Work.fCalc[7] - #Work.fCmdVirSpeed) + 1);
               #Work.fVirSpeedLog := #Work.fCalc[7] + (#Work.fCmdVirSpeed - #Work.fCalc[7]) * (1 / (1 + EXP(- (#Work.fCalc[0] * #fSlopeDecLog - #Cfg.fFirstStepNepero))));
           END_IF;
           #Work.fCalc[4] := 0;
       ELSE
           IF #Work.fVirSpeedLog > 0 THEN
               #Work.fCalc[4] := #Work.fCalc[4] + #DataIn.ifTimeScan;
           END_IF;
           #fSlopeDecLog := (12 * #Work.fDecOnWork) / (#Work.fCalc[5] + 1);
           #Work.fVirSpeedLog := #Work.fCalc[5] * (1 - (1 / (1 + EXP(- ((#Work.fCalc[4]) * #fSlopeDecLog - #Cfg.fFirstStepNepero)))));
           #Work.fCalc[10] := #Work.fCalc[5];
           #Work.fCalc[7] := #Work.fVirSpeedLog;
           #Work.fCalc[0] := 0;
       END_IF;


       IF NOT (#DataIn.ixEnablePos) AND (#Work.fVirSpeedLog < 1.0) THEN
           #Work.xCalc[0] := TRUE;
       END_IF;

       IF #Work.xStopVirPositioner OR #Work.xEnablePulse OR #Work.xCalc[0] THEN
           #Work.fVirSpeed := 0;
           #Work.fCalc[0] := 0;
           #Work.fCalc[4] := 0;
           #Work.fCalc[5] := 0;
           #Work.fCalc[7] := 0;
           #Work.fCalc[10] := 0;
        END_IF;

   END_IF;
END_REGION

REGION Network 14 (SCL): Calcolo Profilo velocità posizionatore COSENO
   // Calcolo velocità profilo posizionatore.
   // Durante la fase di fermata modulo la decelerazione per fermarmi nella posizione 
   // richiesta; la variazione massima di decelerazione è del 50%. Questo è 
   // necessario in quanto il punto di richiesta velocità 0 è afflitto dall'errore 
   // generato dal tempo di scansione della CPU.
   IF #Work."xCurveS-L" THEN
       IF #Work.fCmdVirSpeed > 0 THEN
           #Work.fCalc[19] := #Work.fCalc[19] + #DataIn.ifTimeScan;
                   #Work.fCalc[13] := 1;
                   IF #Work.fCalc[13] < #Work.fVirSpeedCos THEN
                       #Work.fCalc[13] := #Work.fVirSpeedCos;
                   END_IF;
                   #fSlopeAccCos := #PiGrego / ((ABS(#Work.fCmdVirSpeed - #Work.fCalc[17]) + 1) / #Work.fAccOnWork);
                   IF NOT #Work.xCmdVirSpeedChanged THEN
                       IF #fSlopeAccCos * #Work.fCalc[19] < #PiGrego THEN
                           #Work.fVirSpeedCos := #Work.fCalc[17] + (#Work.fCmdVirSpeed - #Work.fCalc[17]) * 0.5 * (COS(#fSlopeAccCos * #Work.fCalc[19] + #PiGrego) + 1);
                       ELSE
                           #Work.fVirSpeedCos := #Work.fCmdVirSpeed;
                       END_IF;
                   ELSE
                       #fSlopeDecCos := #PiGrego / ((ABS(#Work.fCmdVirSpeed - #Work.fCalc[17]) + 1) / #Work.fDecOnWork);
                       IF #fSlopeDecCos * #Work.fCalc[19] < #PiGrego THEN
                           #Work.fVirSpeedCos := #Work.fCalc[17] + (#Work.fCmdVirSpeed - #Work.fCalc[17]) * 0.5 * (COS(#fSlopeDecCos * #Work.fCalc[19] + #PiGrego) + 1);
                       ELSE
                           #Work.fVirSpeedCos := #Work.fCmdVirSpeed;
                       END_IF;

                   END_IF;
                   #Work.fCalc[18] := #DataIn.ifTimeScan * 0;
           ELSE
               #Work.fCalc[19] := 0;
               IF #Work.fVirSpeedCos > 0 THEN
                   #Work.fCalc[18] := #Work.fCalc[18] + #DataIn.ifTimeScan;
                   #fSlopeDecCos := #PiGrego / (#Work.fCalc[13] / #Work.fDecOnWork);
                   IF #fSlopeDecCos * #Work.fCalc[18] < #PiGrego THEN
                       #Work.fVirSpeedCos := #Work.fCalc[13] * 0.5 * (COS(#fSlopeDecCos * #Work.fCalc[18]) + 1);
                   ELSE
                       #Work.fVirSpeedCos := 0;
                   END_IF;
                   #Work.fCalc[17] := #Work.fVirSpeedCos;
                   #Work.fCalc[19] := 0;
               END_IF;
       END_IF;

           IF #Work.xStopVirPositioner OR #Work.xEnablePulse THEN
               #Work.fVirSpeed := 0;
               #Work.fVirSpeedCos := 0;
               #Work.fCalc[13] := 0;
               #Work.fCalc[17] := 0;
               #Work.fCalc[18] := 0;
               #Work.fCalc[19] := 0;
           END_IF;
   END_IF;
END_REGION

REGION Network 15 (SCL): Gestione profilo posizionatore
   IF NOT #Work.xStopVirPositioner THEN
       CASE #Cfg."xCurveS-L" OF
           0:
               #Work.fVirSpeed := #Work.fVirSpeedLinear;
           1:
               IF #Work."xCurveS-L" THEN
                   IF #Work.fVirSpeedLog >= 1 THEN
                       #Work.fVirSpeed := #Work.fVirSpeedLog;
                   ELSE
                       #Work.fVirSpeed := 0;
                   END_IF;
               ELSE
                   #Work.fVirSpeed := #Work.fVirSpeedLinear;
               END_IF;
           2:
               #Work.fVirSpeed := #Work.fVirSpeedCos;
       END_CASE;

       IF (#Work.fVirSpeed < #Cfg.fMinSpeed) AND #Work.xINEnable AND NOT (#DataOut.oxPosError) AND #Work.xDriveReady THEN
           #Work.fVirSpeed := #Cfg.fMinSpeed;
       END_IF;

       IF #DataIn.ixEnableLevRes AND #DataIn.ixLevelReached AND #Work.fVirSpeed = #Cfg.fMinSpeed THEN
           #Work.fVirSpeed := 0;
       END_IF;

   ELSE
       #Work.xCmdVirSpeedChanged := FALSE;
   END_IF;
END_REGION

REGION Network 16 (SCL): Calcolo posizione con legge di moto
   // Calcolo la posizione del generatore di profilo sul tempo 
   // di scansione della CPU.
   IF NOT #Work.xStopVirPositioner AND ((#DataIn.ixEnableLevRes AND NOT #DataIn.ixLevelReached OR NOT #DataIn.ixEnableLevRes))
       AND ( #Work.xDecStop OR  NOT (#Work.xCalc[13])) THEN
       IF #Work.f_PositionTarget > #Work.fVirPos THEN
           #Work.fVirPos := #Work.fVirPos + (#Work.fVirSpeed * #DataIn.ifTimeScan);
       ELSE
           #Work.fVirPos := #Work.fVirPos - (#Work.fVirSpeed * #DataIn.ifTimeScan);
       END_IF;
   END_IF;
END_REGION

REGION Network 17: Memo start pos
   RUNG wire#powerrail
      { S7_Templates := "SrcType := Real" } GT_Contact(in1 := #Work.fOutSpeedMot, in2 := 0.0)
      P_Trig( #Work.xCalc[20] )
      Move(in := #DataIn.ifEncoder, out1 => #Work.fCalc[20])
      R_Coil( #Work.xDecStop )
      Coil( #Work.xEnablePulse )
   END_RUNG
   // the same network as SCL:
   #_w1 := #Work.fOutSpeedMot > 0.0;
   #_w2 := #_w1 AND NOT #Work.xCalc[20];   // rising edge
   #Work.xCalc[20] := #_w1;
   IF #_w2 THEN
       #Work.fCalc[20] := #DataIn.ifEncoder;
       #Work.xDecStop := FALSE;
   END_IF;
   #Work.xEnablePulse := #_w2;
END_REGION

REGION Network 18 (SCL): Calcolo spazio di arresto del profilo con dati attuali
   #DataOut.ofSpaceStop := #Cfg.fMotWindPos + #Cfg.fMotAdvStopPosition + (SQR(#Work.fVirSpeed)) / (#Work.fDecOnWork * 2.0);
   IF (ABS(#Work.f_PositionTarget - #Work.fVirPos)) <= #DataOut.ofSpaceStop AND NOT #Work.xDecStop THEN
       #Work.xCalc[13] := 1;
   ELSE
       #Work.xCalc[13] := 0;
   END_IF;

   IF NOT #Cfg.xDisablePos THEN
       #DataOut.ofSpaceStop := #Cfg.fMotWindPos + #Cfg.fMotAdvStopPosition + (SQR(#Work.fVirSpeed)) / (#Work.fDecOnWork * 2.0);
   ELSE
       #DataOut.ofSpaceStop := #Cfg.fMotWindPos + #Cfg.fMotAdvStopPosition + (SQR(#DataOut.ofSpeedRequest)) / (#Work.fDecOnWork * 2.0);
   END_IF;




   IF #DataIn.ixEnableLevRes AND #Work.xDecResearch  THEN
       #DataOut.ofSpaceStop := #Cfg.fMotWindPos + #Cfg.fMotAdvStopPosition + (SQR(#DataIn.ifSpeedLev)) / (#Work.fDecOnWork * 2.0);
   END_IF;

   #DataOut.ofSpaceStart := (SQR(#Work.f_SpeedReqCalc)) / (#Work.fAccOnWork * 2.0);
   #DataOut.ofSpaceLevRes := (SQR(#Work.fVirSpeed) / (#Work.fDecOnWork * 2.0)) - (SQR( #DataIn.ifSpeedLev) / (#Work.fDecOnWork * 2.0)) + 50;
   #DataOut.oxAccOnWork := ABS(#Work.fCalc[20] - #DataIn.ifEncoder) < #DataOut.ofSpaceStart;
   #DataOut.oxDecOnWork := #Work.xDecStop OR ((#Work.fOutSpeedMot > 0) AND NOT #Work.xINEnable);

   IF NOT #Cfg.xDisablePos THEN
       IF (ABS(#Work.f_PositionTarget - #Work.fVirPos)) <= #DataOut.ofSpaceStop THEN
           #Work.xDecStop := 1;
       END_IF;
   ELSE
       IF (ABS(#Work.f_PositionTarget - #DataIn.ifEncoder)) <= #DataOut.ofSpaceStop THEN
           #Work.xDecStop := 1;
       END_IF;
   END_IF;

   // IF NOT (#Work.xEnablePos) OR (#Work.xStopVirPositioner AND NOT (#Cfg.xDisablePos))
   //     OR (#DataOut.oxEndPos AND #Cfg.xDisablePos)THEN
   //     #Work.xDecStop := 0;
   // END_IF;
   // test
   IF NOT (#Work.xEnablePos) THEN
       #Work.xDecStop := 0;
   END_IF;

   IF #DataIn.ixEnableLevRes AND #Work.xINEnable AND NOT #DataOut.oxEndPos AND #DataOut.ofSpeedRequest > 0 THEN
       IF #DataOut.oxCmdMotorBack AND (#DataIn.ifEncoder < (#DataIn.ifPositionStartLev + #DataOut.ofSpaceLevRes + 1)) OR
           #DataOut.oxCmdMotorForw AND (#DataIn.ifEncoder > (#DataIn.ifPositionStartLev - #DataOut.ofSpaceLevRes - 1))  THEN
           #Work.xDecResearch := 1;
       END_IF;
   END_IF;

   IF NOT #DataIn.ixEnableLevRes THEN
       #Work.xDecResearch := 0;
   END_IF;
END_REGION

REGION Network 19: Reset arresto posizionatore virtuale
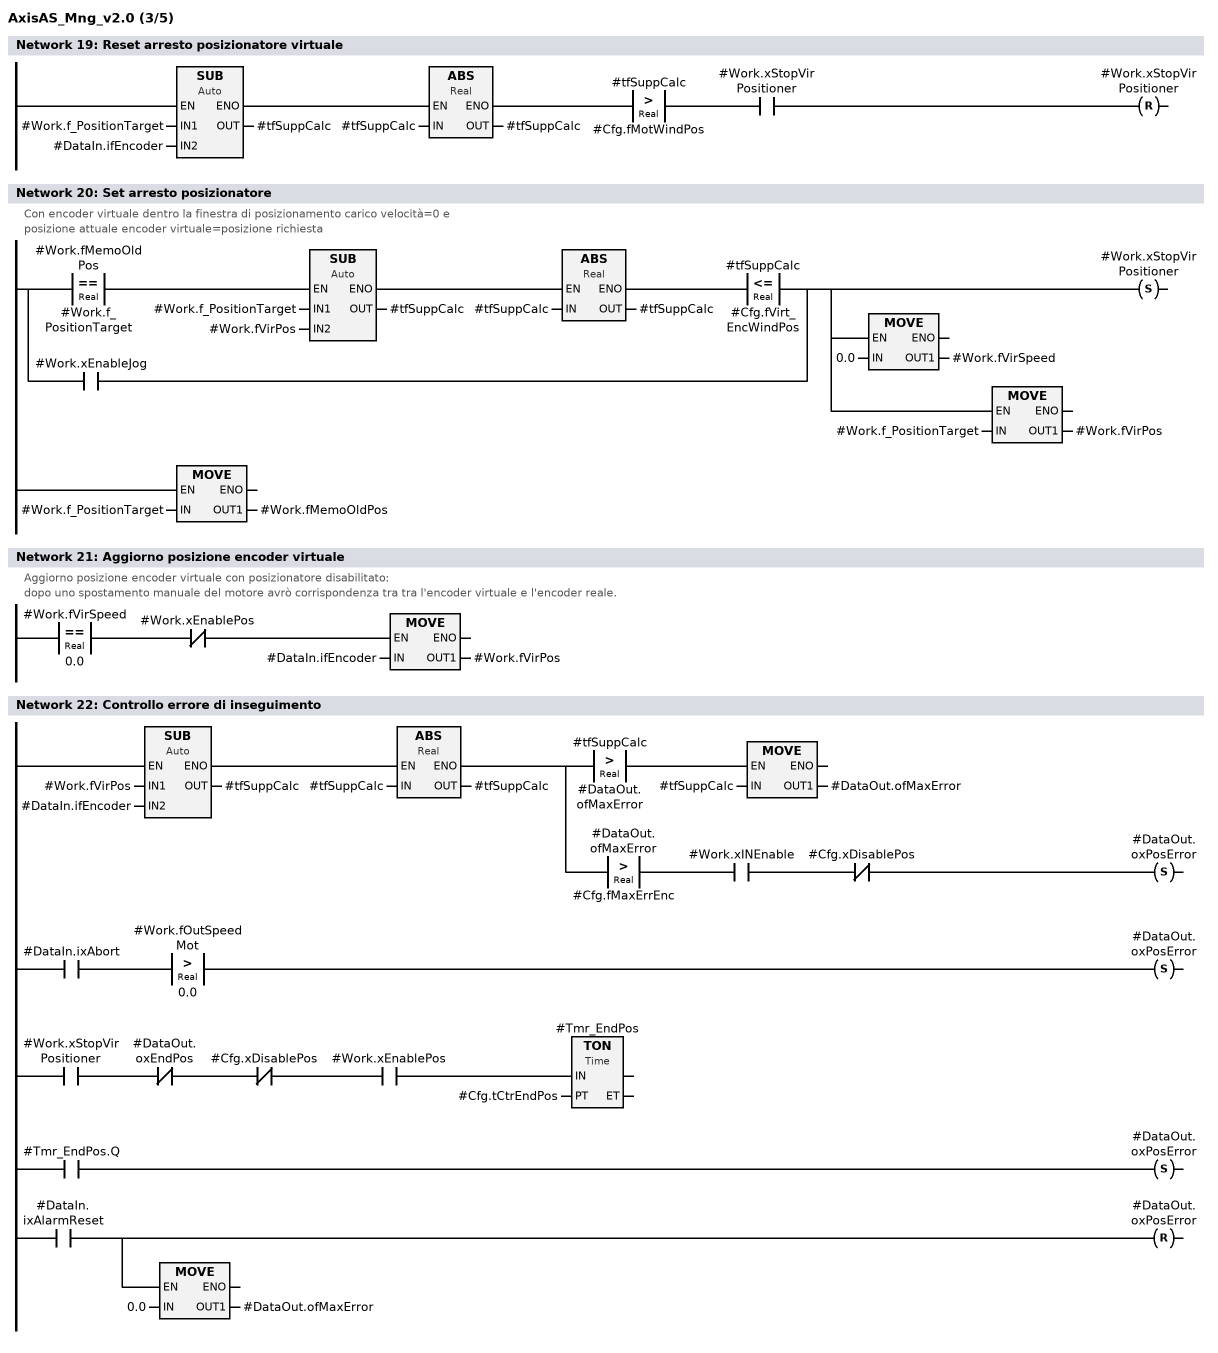
   RUNG wire#powerrail
      Sub(in1 := #Work.f_PositionTarget, in2 := #DataIn.ifEncoder, out => #tfSuppCalc)
      { S7_Templates := "SrcType := Real" } Abs(in := #tfSuppCalc, out => #tfSuppCalc)
      { S7_Templates := "SrcType := Real" } GT_Contact(in1 := #tfSuppCalc, in2 := #Cfg.fMotWindPos)
      Contact( #Work.xStopVirPositioner )
      R_Coil( #Work.xStopVirPositioner )
   END_RUNG
   // the same network as SCL:
   #tfSuppCalc := #Work.f_PositionTarget - #DataIn.ifEncoder;
   #tfSuppCalc := ABS(#tfSuppCalc);
   IF (#tfSuppCalc > #Cfg.fMotWindPos) AND #Work.xStopVirPositioner THEN
       #Work.xStopVirPositioner := FALSE;
   END_IF;
END_REGION

REGION Network 20: Set arresto posizionatore
   // Con encoder virtuale dentro la finestra di posizionamento carico velocità=0 e 
   // posizione attuale encoder virtuale=posizione richiesta
   RUNG wire#powerrail
      { S7_Templates := "SrcType := Real" } EQ_Contact(in1 := #Work.fMemoOldPos, in2 := #Work.f_PositionTarget)
      Sub(in1 := #Work.f_PositionTarget, in2 := #Work.fVirPos, out => #tfSuppCalc)
      { S7_Templates := "SrcType := Real" } Abs(in := #tfSuppCalc, out => #tfSuppCalc)
      { S7_Templates := "SrcType := Real" } LE_Contact(in1 := #tfSuppCalc, in2 := #Cfg.fVirt_EncWindPos)
      wire#w1
      S_Coil( #Work.xStopVirPositioner )
   END_RUNG
   RUNG wire#powerrail
      Contact( #Work.xEnableJog )
   END_RUNG wire#w1
   RUNG wire#w1
      Move(in := 0.0, out1 => #Work.fVirSpeed)
   END_RUNG
   RUNG wire#w1
      Move(in := #Work.f_PositionTarget, out1 => #Work.fVirPos)
   END_RUNG
   RUNG wire#powerrail
      Move(in := #Work.f_PositionTarget, out1 => #Work.fMemoOldPos)
   END_RUNG
   // the same network as SCL:
   #_w1 := #Work.fMemoOldPos = #Work.f_PositionTarget;
   IF #_w1 THEN
       #tfSuppCalc := #Work.f_PositionTarget - #Work.fVirPos;
       #tfSuppCalc := ABS(#tfSuppCalc);
   END_IF;
   IF (#_w1 AND (#tfSuppCalc <= #Cfg.fVirt_EncWindPos)) OR #Work.xEnableJog THEN
       #Work.xStopVirPositioner := TRUE;
       #Work.fVirSpeed := 0.0;
       #Work.fVirPos := #Work.f_PositionTarget;
   END_IF;
   #Work.fMemoOldPos := #Work.f_PositionTarget;
END_REGION

REGION Network 21: Aggiorno posizione encoder virtuale
   // Aggiorno posizione encoder virtuale con posizionatore disabilitato: 
   // dopo uno spostamento manuale del motore avrò corrispondenza tra tra l'encoder virtuale e l'encoder reale.
   RUNG wire#powerrail
      { S7_Templates := "SrcType := Real" } EQ_Contact(in1 := #Work.fVirSpeed, in2 := 0.0)
      I_Contact( #Work.xEnablePos )
      Move(in := #DataIn.ifEncoder, out1 => #Work.fVirPos)
   END_RUNG
   // the same network as SCL:
   IF (#Work.fVirSpeed = 0.0) AND NOT #Work.xEnablePos THEN #Work.fVirPos := #DataIn.ifEncoder; END_IF;
END_REGION

REGION Network 22: Controllo errore di inseguimento
   RUNG wire#powerrail
      Sub(in1 := #Work.fVirPos, in2 := #DataIn.ifEncoder, out => #tfSuppCalc)
      { S7_Templates := "SrcType := Real" } Abs(in := #tfSuppCalc, out => #tfSuppCalc)
      wire#w1
      { S7_Templates := "SrcType := Real" } GT_Contact(in1 := #tfSuppCalc, in2 := #DataOut.ofMaxError)
      Move(in := #tfSuppCalc, out1 => #DataOut.ofMaxError)
   END_RUNG
   RUNG wire#w1
      { S7_Templates := "SrcType := Real" } GT_Contact(in1 := #DataOut.ofMaxError, in2 := #Cfg.fMaxErrEnc)
      Contact( #Work.xINEnable )
      I_Contact( #Cfg.xDisablePos )
      S_Coil( #DataOut.oxPosError )
   END_RUNG
   RUNG wire#powerrail
      Contact( #DataIn.ixAbort )
      { S7_Templates := "SrcType := Real" } GT_Contact(in1 := #Work.fOutSpeedMot, in2 := 0.0)
      S_Coil( #DataOut.oxPosError )
   END_RUNG
   RUNG wire#powerrail
      Contact( #Work.xStopVirPositioner )
      I_Contact( #DataOut.oxEndPos )
      I_Contact( #Cfg.xDisablePos )
      Contact( #Work.xEnablePos )
      { S7_Templates := "time_type := Time" } #Tmr_EndPos.TON(pt := #Cfg.tCtrEndPos, et =>)
   END_RUNG
   RUNG wire#powerrail
      Contact( #Tmr_EndPos.Q )
      S_Coil( #DataOut.oxPosError )
   END_RUNG
   RUNG wire#powerrail
      Contact( #DataIn.ixAlarmReset )
      wire#w2
      R_Coil( #DataOut.oxPosError )
   END_RUNG
   RUNG wire#w2
      Move(in := 0.0, out1 => #DataOut.ofMaxError)
   END_RUNG
   // the same network as SCL:
   #tfSuppCalc := #Work.fVirPos - #DataIn.ifEncoder;
   #tfSuppCalc := ABS(#tfSuppCalc);
   IF #tfSuppCalc > #DataOut.ofMaxError THEN #DataOut.ofMaxError := #tfSuppCalc; END_IF;
   IF (#DataOut.ofMaxError > #Cfg.fMaxErrEnc) AND #Work.xINEnable AND NOT #Cfg.xDisablePos THEN
       #DataOut.oxPosError := TRUE;
   END_IF;
   IF #DataIn.ixAbort AND (#Work.fOutSpeedMot > 0.0) THEN #DataOut.oxPosError := TRUE; END_IF;
   #Tmr_EndPos.TON(IN := #Work.xStopVirPositioner AND NOT #DataOut.oxEndPos AND NOT #Cfg.xDisablePos AND #Work.xEnablePos,
                   PT := #Cfg.tCtrEndPos);
   IF #Tmr_EndPos.Q THEN #DataOut.oxPosError := TRUE; END_IF;
   IF #DataIn.ixAlarmReset THEN
       #DataOut.oxPosError := FALSE;
       #DataOut.ofMaxError := 0.0;
   END_IF;
END_REGION

REGION Network 23 (SCL): Calcolo correzione PID
   #Work."fLim+Ppid" :=   (#Cfg.fMaxSpeed * 0.2);
   #Work."fLim-Ppid" := - (#Cfg.fMaxSpeed * 0.2);
   // test  ... limitare azione correttiva non su max speed ma su actual speed ??
   // #Work."fLim+Ppid" :=   ( #Work.fVirSpeed * 0.2);
   // #Work."fLim-Ppid" := - ( #Work.fVirSpeed * 0.2);

   IF (#DataIn.ixEnableLevRes AND #Work.xDecResearch AND NOT #Work.xDecStop) OR #DataOut.oxEndPos OR (NOT #Work.xEnablePos)
       OR NOT(#Work.xINEnable)  THEN
       #Work.fMemoMaxSpeed := 1;
   END_IF;

   IF (ABS(#Work.fVirSpeed) > #Work.fMemoMaxSpeed) THEN
       #Work.fMemoMaxSpeed := #Work.fVirSpeed;
   END_IF;
   #Work.fSuppCalcPpid := ((#Work.fMemoMaxSpeed - #Work.fVirSpeed) / #Work.fMemoMaxSpeed) * #Cfg.fKPpidDec_Pos + #Cfg.fKPpid_Pos;
END_REGION

REGION Network 24 (SCL): Amplifico correzione PID a piramide su posizionamento
   #Work.fPpid := (#Work.fVirPos -  #DataIn.ifEncoder) * #Work.fSuppCalcPpid;
   IF #DataOut.oxCmdMotorBack THEN
       #Work.fPpid := - (#Work.fVirPos -  #DataIn.ifEncoder) * #Work.fSuppCalcPpid;
   END_IF;

   IF #Work.fPpid > #Work."fLim+Ppid" THEN
       #Work.fPpid := #Work."fLim+Ppid";
   END_IF;
   IF #Work.fPpid < #Work."fLim-Ppid" THEN
       #Work.fPpid := #Work."fLim-Ppid";
   END_IF;

   IF NOT #Work.xEnablePos OR #Work.xStopVirPositioner OR #DataOut.oxPosError OR #Cfg.xDisablePos THEN
       #Work.fPpid := 0;
   END_IF;
END_REGION

REGION Network 25 (SCL): Carico velocità per motore da jog o posizionatore
   #Work.fOutSpeedMot := 0.0;
   IF #Work.xEnablePos THEN // test AND ((#DataIn.ixEnableLevRes AND NOT #DataIn.ixLevelReached) OR NOT #DataIn.ixEnableLevRes)  THEN
       IF (ABS(#DataIn.ifEncoder - #Work.f_PositionTarget) >= #Cfg.fMotWindPos) THEN
           IF #Work.fVirSpeed + #Work.fPpid <= 0 THEN
               #Work.fOutSpeedMot := #Work.fVirSpeed/2;
           ELSE
               #Work.fOutSpeedMot := #Work.fVirSpeed + #Work.fPpid;
           END_IF;
       END_IF;
       IF NOT #DataOut.oxEndPos AND #Work.xDecStop AND (#Work.fVirSpeed = 0) AND #Work.xINEnable AND (ABS(#DataIn.ifEncoder - #Work.f_PositionTarget) >= #Cfg.fMotWindPos)
           OR (ABS(#DataIn.ifEncoder - #Work.f_PositionTarget) >= #Cfg.fMotWindPos) AND (#Work.fOutSpeedMot < #Cfg.fMinSpeed)
           AND #Work.xINEnable AND #Work.xDriveReady AND ((#DataIn.ixEnableLevRes AND NOT #DataIn.ixLevelReached) OR NOT #DataIn.ixEnableLevRes)
       THEN
           #Work.fOutSpeedMot := #Cfg.fMinSpeed;
       END_IF;
   END_IF;

   IF  #Work.xEnableJog THEN
       #Work.fOutSpeedMot := #Work.fJogSpeed;
   END_IF;
END_REGION

REGION Network 26 (SCL): Out velocità motore
   IF #Work.fOutSpeedMot > 0.0 AND NOT( #DataIn.ixAbort) AND (NOT(#DataOut.oxEndPos) OR  #Work.xEnableJog) THEN
       #DataOut.ofSpeedRequest := #Work.fOutSpeedMot;
       IF #Work.fOutSpeedMot < #Cfg.fMinSpeed AND NOT (#DataOut.oxPosError) THEN
           #DataOut.ofSpeedRequest := #Cfg.fMinSpeed;
       END_IF;
       IF #Work.fOutSpeedMot > #Cfg.fMaxSpeed  THEN
           #DataOut.ofSpeedRequest := #Cfg.fMaxSpeed;
       END_IF;
   ELSE
       #DataOut.ofSpeedRequest := 0;
   END_IF;
END_REGION

REGION Network 27 (SCL): OUT Conferma posizionamento eseguito (velocità stop)
   IF #DataOut.ofSpeedRequest = 0 THEN
       #DataOut.oxStopSpeed := TRUE;
   ELSE
       #DataOut.oxStopSpeed := FALSE;
   END_IF;

   #DataOut.ofEncMotorPos := #DataIn.ifEncoder;
END_REGION

REGION Network 28: OUT Conferma posizionamento eseguito (posizionamento terminato) + Camma posizione allargata
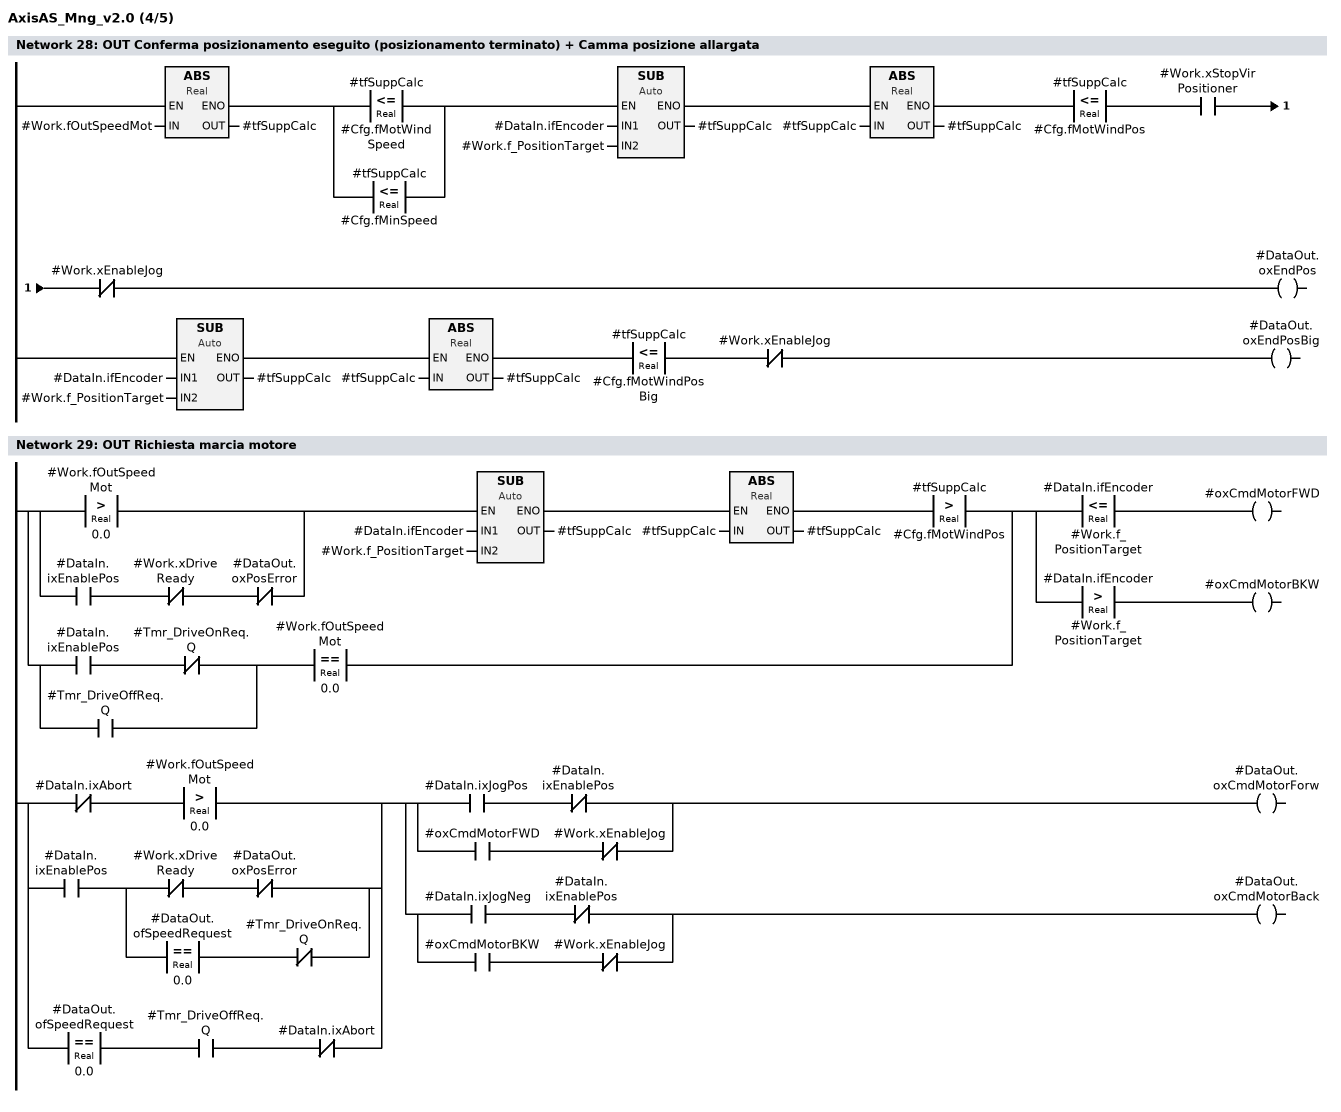
   RUNG wire#powerrail
      { S7_Templates := "SrcType := Real" } Abs(in := #Work.fOutSpeedMot, out => #tfSuppCalc)
      wire#w1
      { S7_Templates := "SrcType := Real" } LE_Contact(in1 := #tfSuppCalc, in2 := #Cfg.fMotWindSpeed)
      wire#w2
      Sub(in1 := #DataIn.ifEncoder, in2 := #Work.f_PositionTarget, out => #tfSuppCalc)
      { S7_Templates := "SrcType := Real" } Abs(in := #tfSuppCalc, out => #tfSuppCalc)
      { S7_Templates := "SrcType := Real" } LE_Contact(in1 := #tfSuppCalc, in2 := #Cfg.fMotWindPos)
      Contact( #Work.xStopVirPositioner )
      I_Contact( #Work.xEnableJog )
      Coil( #DataOut.oxEndPos )
   END_RUNG
   RUNG wire#w1
      { S7_Templates := "SrcType := Real" } LE_Contact(in1 := #tfSuppCalc, in2 := #Cfg.fMinSpeed)
   END_RUNG wire#w2
   RUNG wire#powerrail
      Sub(in1 := #DataIn.ifEncoder, in2 := #Work.f_PositionTarget, out => #tfSuppCalc)
      { S7_Templates := "SrcType := Real" } Abs(in := #tfSuppCalc, out => #tfSuppCalc)
      { S7_Templates := "SrcType := Real" } LE_Contact(in1 := #tfSuppCalc, in2 := #Cfg.fMotWindPosBig)
      I_Contact( #Work.xEnableJog )
      Coil( #DataOut.oxEndPosBig )
   END_RUNG
   // the same network as SCL:
   #tfSuppCalc := ABS(#Work.fOutSpeedMot);
   #_w1 := (#tfSuppCalc <= #Cfg.fMotWindSpeed) OR (#tfSuppCalc <= #Cfg.fMinSpeed);
   IF #_w1 THEN
       #tfSuppCalc := #DataIn.ifEncoder - #Work.f_PositionTarget;
       #tfSuppCalc := ABS(#tfSuppCalc);
   END_IF;
   #DataOut.oxEndPos := #_w1 AND (#tfSuppCalc <= #Cfg.fMotWindPos) AND #Work.xStopVirPositioner AND NOT #Work.xEnableJog;
   #tfSuppCalc := #DataIn.ifEncoder - #Work.f_PositionTarget;
   #tfSuppCalc := ABS(#tfSuppCalc);
   #DataOut.oxEndPosBig := (#tfSuppCalc <= #Cfg.fMotWindPosBig) AND NOT #Work.xEnableJog;
END_REGION

REGION Network 29: OUT Richiesta marcia motore
   RUNG wire#powerrail
      { S7_Templates := "SrcType := Real" } GT_Contact(in1 := #Work.fOutSpeedMot, in2 := 0.0)
      wire#w1
      Sub(in1 := #DataIn.ifEncoder, in2 := #Work.f_PositionTarget, out => #tfSuppCalc)
      { S7_Templates := "SrcType := Real" } Abs(in := #tfSuppCalc, out => #tfSuppCalc)
      { S7_Templates := "SrcType := Real" } GT_Contact(in1 := #tfSuppCalc, in2 := #Cfg.fMotWindPos)
      wire#w2
      { S7_Templates := "SrcType := Real" } LE_Contact(in1 := #DataIn.ifEncoder, in2 := #Work.f_PositionTarget)
      Coil( #oxCmdMotorFWD )
   END_RUNG
   RUNG wire#powerrail
      Contact( #DataIn.ixEnablePos )
      I_Contact( #Work.xDriveReady )
      I_Contact( #DataOut.oxPosError )
   END_RUNG wire#w1
   RUNG wire#powerrail
      Contact( #DataIn.ixEnablePos )
      I_Contact( #Tmr_DriveOnReq.Q )
      wire#w3
      { S7_Templates := "SrcType := Real" } EQ_Contact(in1 := #Work.fOutSpeedMot, in2 := 0.0)
   END_RUNG wire#w2
   RUNG wire#powerrail
      Contact( #Tmr_DriveOffReq.Q )
   END_RUNG wire#w3
   RUNG wire#w2
      { S7_Templates := "SrcType := Real" } GT_Contact(in1 := #DataIn.ifEncoder, in2 := #Work.f_PositionTarget)
      Coil( #oxCmdMotorBKW )
   END_RUNG
   RUNG wire#powerrail
      I_Contact( #DataIn.ixAbort )
      { S7_Templates := "SrcType := Real" } GT_Contact(in1 := #Work.fOutSpeedMot, in2 := 0.0)
      wire#w4
      Contact( #DataIn.ixJogPos )
      I_Contact( #DataIn.ixEnablePos )
      wire#w6
      Coil( #DataOut.oxCmdMotorForw )
   END_RUNG
   RUNG wire#powerrail
      Contact( #DataIn.ixEnablePos )
      wire#w5
      I_Contact( #Work.xDriveReady )
      I_Contact( #DataOut.oxPosError )
   END_RUNG wire#w4
   RUNG wire#w5
      { S7_Templates := "SrcType := Real" } EQ_Contact(in1 := #DataOut.ofSpeedRequest, in2 := 0.0)
      I_Contact( #Tmr_DriveOnReq.Q )
   END_RUNG wire#w4
   RUNG wire#powerrail
      { S7_Templates := "SrcType := Real" } EQ_Contact(in1 := #DataOut.ofSpeedRequest, in2 := 0.0)
      Contact( #Tmr_DriveOffReq.Q )
      I_Contact( #DataIn.ixAbort )
   END_RUNG wire#w4
   RUNG wire#w4
      Contact( #oxCmdMotorFWD )
      I_Contact( #Work.xEnableJog )
   END_RUNG wire#w6
   RUNG wire#w4
      Contact( #DataIn.ixJogNeg )
      I_Contact( #DataIn.ixEnablePos )
      wire#w7
      Coil( #DataOut.oxCmdMotorBack )
   END_RUNG
   RUNG wire#w4
      Contact( #oxCmdMotorBKW )
      I_Contact( #Work.xEnableJog )
   END_RUNG wire#w7
   // the same network as SCL:
   #_w1 := (#Work.fOutSpeedMot > 0.0) OR (#DataIn.ixEnablePos AND NOT #Work.xDriveReady AND NOT #DataOut.oxPosError);
   IF #_w1 THEN
       #tfSuppCalc := #DataIn.ifEncoder - #Work.f_PositionTarget;
       #tfSuppCalc := ABS(#tfSuppCalc);
   END_IF;
   #_w2 := (#_w1 AND (#tfSuppCalc > #Cfg.fMotWindPos)) OR (((#DataIn.ixEnablePos AND NOT #Tmr_DriveOnReq.Q) OR #Tmr_DriveOffReq.Q) AND (#Work.fOutSpeedMot = 0.0));
   #oxCmdMotorFWD := #_w2 AND (#DataIn.ifEncoder <= #Work.f_PositionTarget);
   #oxCmdMotorBKW := #_w2 AND (#DataIn.ifEncoder > #Work.f_PositionTarget);
   #_w3 := (NOT #DataIn.ixAbort AND (#Work.fOutSpeedMot > 0.0)) OR (#DataIn.ixEnablePos AND ((NOT #Work.xDriveReady AND NOT #DataOut.oxPosError) OR ((#DataOut.ofSpeedRequest = 0.0) AND NOT #Tmr_DriveOnReq.Q))) OR ((#DataOut.ofSpeedRequest = 0.0) AND #Tmr_DriveOffReq.Q AND NOT #DataIn.ixAbort);
   #DataOut.oxCmdMotorForw := #_w3 AND ((#DataIn.ixJogPos AND NOT #DataIn.ixEnablePos) OR (#oxCmdMotorFWD AND NOT #Work.xEnableJog));
   #DataOut.oxCmdMotorBack := #_w3 AND ((#DataIn.ixJogNeg AND NOT #DataIn.ixEnablePos) OR (#oxCmdMotorBKW AND NOT #Work.xEnableJog));
END_REGION

REGION Network 30: OUT freno motore
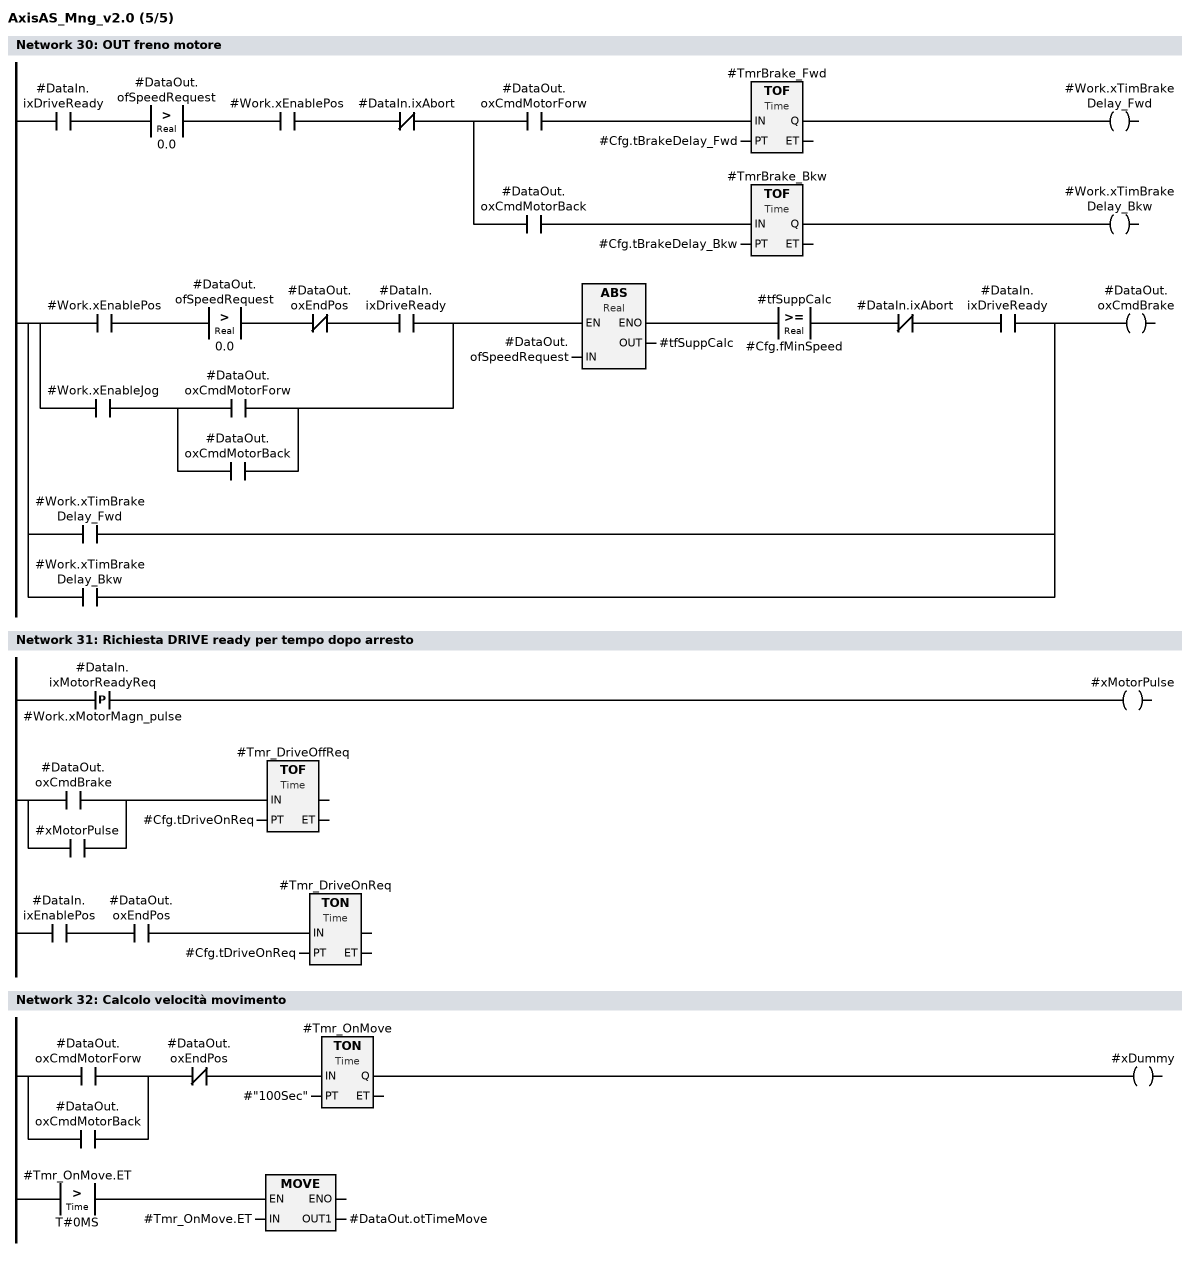
   RUNG wire#powerrail
      Contact( #DataIn.ixDriveReady )
      { S7_Templates := "SrcType := Real" } GT_Contact(in1 := #DataOut.ofSpeedRequest, in2 := 0.0)
      Contact( #Work.xEnablePos )
      I_Contact( #DataIn.ixAbort )
      wire#w1
      Contact( #DataOut.oxCmdMotorForw )
      { S7_Templates := "time_type := Time" } #TmrBrake_Fwd.TOF(pt := #Cfg.tBrakeDelay_Fwd, et =>)
      Coil( #Work.xTimBrakeDelay_Fwd )
   END_RUNG
   RUNG wire#w1
      Contact( #DataOut.oxCmdMotorBack )
      { S7_Templates := "time_type := Time" } #TmrBrake_Bkw.TOF(pt := #Cfg.tBrakeDelay_Bkw, et =>)
      Coil( #Work.xTimBrakeDelay_Bkw )
   END_RUNG
   RUNG wire#powerrail
      Contact( #Work.xEnablePos )
      { S7_Templates := "SrcType := Real" } GT_Contact(in1 := #DataOut.ofSpeedRequest, in2 := 0.0)
      I_Contact( #DataOut.oxEndPos )
      Contact( #DataIn.ixDriveReady )
      wire#w2
      { S7_Templates := "SrcType := Real" } Abs(in := #DataOut.ofSpeedRequest, out => #tfSuppCalc)
      { S7_Templates := "SrcType := Real" } GE_Contact(in1 := #tfSuppCalc, in2 := #Cfg.fMinSpeed)
      I_Contact( #DataIn.ixAbort )
      Contact( #DataIn.ixDriveReady )
      wire#w4
      Coil( #DataOut.oxCmdBrake )
   END_RUNG
   RUNG wire#powerrail
      Contact( #Work.xEnableJog )
      wire#w3
      Contact( #DataOut.oxCmdMotorForw )
   END_RUNG wire#w2
   RUNG wire#w3
      Contact( #DataOut.oxCmdMotorBack )
   END_RUNG wire#w2
   RUNG wire#powerrail
      Contact( #Work.xTimBrakeDelay_Fwd )
   END_RUNG wire#w4
   RUNG wire#powerrail
      Contact( #Work.xTimBrakeDelay_Bkw )
   END_RUNG wire#w4
   // the same network as SCL:
   #_w1 := #DataIn.ixDriveReady AND (#DataOut.ofSpeedRequest > 0.0) AND #Work.xEnablePos AND NOT #DataIn.ixAbort;
   #TmrBrake_Fwd.TOF(IN := #_w1 AND #DataOut.oxCmdMotorForw, PT := #Cfg.tBrakeDelay_Fwd);
   #Work.xTimBrakeDelay_Fwd := #TmrBrake_Fwd.Q;
   #TmrBrake_Bkw.TOF(IN := #_w1 AND #DataOut.oxCmdMotorBack, PT := #Cfg.tBrakeDelay_Bkw);
   #Work.xTimBrakeDelay_Bkw := #TmrBrake_Bkw.Q;
   #_w2 := (#Work.xEnablePos AND (#DataOut.ofSpeedRequest > 0.0) AND NOT #DataOut.oxEndPos AND #DataIn.ixDriveReady) OR (#Work.xEnableJog AND (#DataOut.oxCmdMotorForw OR #DataOut.oxCmdMotorBack));
   IF #_w2 THEN #tfSuppCalc := ABS(#DataOut.ofSpeedRequest); END_IF;
   #DataOut.oxCmdBrake := (#_w2 AND (#tfSuppCalc >= #Cfg.fMinSpeed) AND NOT #DataIn.ixAbort AND #DataIn.ixDriveReady) OR #Work.xTimBrakeDelay_Fwd OR #Work.xTimBrakeDelay_Bkw;
END_REGION

REGION Network 31: Richiesta DRIVE ready per tempo dopo arresto
   RUNG wire#powerrail
      P_Contact(operand := #DataIn.ixMotorReadyReq, bit := #Work.xMotorMagn_pulse)
      Coil( #xMotorPulse )
   END_RUNG
   RUNG wire#powerrail
      Contact( #DataOut.oxCmdBrake )
      wire#w1
      { S7_Templates := "time_type := Time" } #Tmr_DriveOffReq.TOF(pt := #Cfg.tDriveOnReq, et =>)
   END_RUNG
   RUNG wire#powerrail
      Contact( #xMotorPulse )
   END_RUNG wire#w1
   RUNG wire#powerrail
      Contact( #DataIn.ixEnablePos )
      Contact( #DataOut.oxEndPos )
      { S7_Templates := "time_type := Time" } #Tmr_DriveOnReq.TON(pt := #Cfg.tDriveOnReq, et =>)
   END_RUNG
   // the same network as SCL:
   #_w1 := #DataIn.ixMotorReadyReq AND NOT #Work.xMotorMagn_pulse;   // rising edge of #DataIn.ixMotorReadyReq
   #Work.xMotorMagn_pulse := #DataIn.ixMotorReadyReq;
   #xMotorPulse := #_w1;
   #Tmr_DriveOffReq.TOF(IN := #DataOut.oxCmdBrake OR #xMotorPulse, PT := #Cfg.tDriveOnReq);
   #Tmr_DriveOnReq.TON(IN := #DataIn.ixEnablePos AND #DataOut.oxEndPos, PT := #Cfg.tDriveOnReq);
END_REGION

REGION Network 32: Calcolo velocità movimento
   RUNG wire#powerrail
      Contact( #DataOut.oxCmdMotorForw )
      wire#w1
      I_Contact( #DataOut.oxEndPos )
      { S7_Templates := "time_type := Time" } #Tmr_OnMove.TON(pt := #"100Sec", et =>)
      Coil( #xDummy )
   END_RUNG
   RUNG wire#powerrail
      Contact( #DataOut.oxCmdMotorBack )
   END_RUNG wire#w1
   RUNG wire#powerrail
      { S7_Templates := "SrcType := Time" } GT_Contact(in1 := #Tmr_OnMove.ET, in2 := T#0MS)
      Move(in := #Tmr_OnMove.ET, out1 => #DataOut.otTimeMove)
   END_RUNG
   // the same network as SCL:
   #Tmr_OnMove.TON(IN := (#DataOut.oxCmdMotorForw OR #DataOut.oxCmdMotorBack) AND NOT #DataOut.oxEndPos,
                   PT := #"100Sec");
   #xDummy := #Tmr_OnMove.Q;
   IF #Tmr_OnMove.ET > T#0MS THEN #DataOut.otTimeMove := #Tmr_OnMove.ET; END_IF;
END_REGION
END_FUNCTION_BLOCK

FUNCTION_BLOCK "AxisAS_Mng"   // FB81, LAD
TITLE = Positioner + PID / Controllo asse + PID
{ S7_Optimized_Access := 'TRUE' }
VERSION : 1.0
// Positioner with Pid management
// 
// Version from master S7: 2.6
// 
// Date: 2017-08-25
// Project: Mora A.
// 
// Version 2.7: -Corrected maximum speed reached in proportional calculation check.
// Version 2.8: -Used Type for CFG data.
// Gestore ASSE per motore asincrono con posizionatore a generazione di profilo ed inseguimento proporzionale + piramidale
// 
// Michele Montanari
// 
// ver 0.0
// - Curva Trapezio
// - Curva "esse" logaritmica
// - Auto gestione curva per piccoli spostamenti
// - Attesa segnale inverter magnetizzato
// 
// ver 1.0 24/01/2023
// - Curva "esse" Coseno
// - Aggiornamneto struttura
// - Calcolo di tutte le curve in simultanea
// - Arresto #Out in posizione su finestra Vir (da provare.... anche su velocità  == 0)
// - Autogestione (selezione) calcolo acc e dec su definizione prestazioni massime
// - Autogestione (selezione) calcolo velocità possibile in funzione del nuovo target
// - Richiesta abilitazione inverter sempre attiva per abbattere tempo di magentizzazione
// - Inversione al volo del moto
// - Gestione interna del freno motore
// stored: MemoryReserve 100, SetENOAutomatically false
   VAR RETAIN
      DataIn : Struct   // Comando asse
         ixEnablePos { S7_SetPoint := 'True'} : Bool;   // Enable positioner / Abilita asse
         ixDriveReady { S7_SetPoint := 'True'} : Bool;   // Inverter magnetizzato
         ixEnableLevRes { S7_SetPoint := 'True'} : Bool;   // Enable level research / Abilita ricerca livello
         ixAlarmReset { S7_SetPoint := 'True'} : Bool;   // Reset alarms / Reset allarmi
         ixAbort { S7_SetPoint := 'True'} : Bool;   // Initializing motor encoder position / Abort sistema
         ixJogPos { S7_SetPoint := 'True'} : Bool;   // Manual Jog positive / Manuale JOG +
         ixJogNeg { S7_SetPoint := 'True'} : Bool;   // Manual Jog negative / Manuale JOG -
         xAutoSpeedDetect { S7_SetPoint := 'True'} : Bool;   // Calcolo velocità automatico su movimento
         xAutoAccDecCalculation { S7_SetPoint := 'True'} : Bool;   // Calcolo Acc Dec automatico su velocità
         ifPositionRequest { S7_SetPoint := 'True'} : Real;   // Position requested (mm) / Quota richiesta (mm)
         ifSpeedRequest { S7_SetPoint := 'True'} : Real;   // Speed requested (mm/sec) / Velocità richiesta (mm/sec)
         ifPositionStartLev { S7_SetPoint := 'True'} : Real;   // Position start research (mm) / Quota inizio ricerca (mm)
         ifSpeedLev { S7_SetPoint := 'True'} : Real;   // Research speed (mm/sec) / Velocità ricerca (mm/sec)
         ifAccRamp { S7_SetPoint := 'True'} : Real;   // Acceleration ramp (mm/sec^2) / * Rampa accelerazione (mm/sec^2)
         ifDecRamp { S7_SetPoint := 'True'} : Real;   // Deceleration ramp (mm/sec^2) / * Rampa decelerazione (mm/sec^2)
         ifTimeScan { S7_SetPoint := 'True'} : Real;   // Time last scan (sec) / Tempo ultima scansione (sec)
         ifEncoder { S7_SetPoint := 'True'} : Real;   // Actual encoder position (encoder) / Posizione attuale encoder
      END_STRUCT;
      DataOut : Struct   // Gestione Inverte e posizioni
         oxCmdMotorForw : Bool;   // Inverter run enabled / Abilitazione marcia Avanti
         oxCmdMotorBack : Bool;   // Abilitazione marcia Indietro
         oxCmdBrake : Bool;   // Enable brake release / Comando stacco freno
         oxPosError { S7_SetPoint := 'True'} : Bool;   // Pursuit error / Allarme: Errore di inseguimento
         oxEndPos : Bool;   // Positioning terminated / Posizionamento terminato
         oxEndPosBig : Bool;   // Posizionamento Allargato terminato
         oxStopSpeed : Bool;   // Motor speed below low limit / Velocità motore = 0
         oxAccOnWork : Bool;   // Rampa Acc in atto
         oxDecOnWork : Bool;   // Rampa Dec in atto
         ofSpeedRequest : Real;   // Motor speed requested (mm/sec) / Velocita motore richiesta (mm/sec)
         ofEncMotorPos : Real;   // Motor encoder position (mm) / Posizione encoder motore (mm)
         ofMaxError : Real;   // Pursuit max error (mm) / Errore massimo di inseguimento (mm)
         ofSpaceStop : Real;   // Stop space requested from current position/speed (mm) / Spazio richiesto per fermata da posizione/velocità attuale (mm)
         ofSpaceLevRes : Real;   // Spazio richiesto per cambio velocità ricerca livello da posizione/velocità attuale (mm)
         ofSpaceStart : Real;   // Spazio richiesto per partenza da posizione/velocità attuale (mm)
         otTimeMove : Time;   // Tempo ultimo movimento
      END_STRUCT;
      Cfg { S7_SetPoint := 'True'} : "AxixAS_CFG_Type";   // Block data initialisation / Configurazione Asse
      Work : Struct   // Positioner management / Gestione Asse
         xEnablePos { S7_SetPoint := 'True'} : Bool;   // Positioner enabled / Posizionatore abilitato/Positioner enabled
         xINEnable : Bool;   // Memo Posizionatore abilitato per inversione
         xDriveReady { S7_SetPoint := 'True'} : Bool;   // Inverter magnetizzato
         xCmdVirSpeedChanged { S7_SetPoint := 'True'} : Bool;   // Variazione target VEL durante missione
         "xCurveS-L" { S7_SetPoint := 'True'} : Bool;   // Curva non lineare
         "xAutoChangeS-L" { S7_SetPoint := 'True'} : Bool;   // Autoimpostazione LIN per brevi spostamenti
         "xCTRAutoChangeS-L" { S7_SetPoint := 'True'} : Bool;   // Autoimpostazione LIN per brevi spostamenti
         xDecStop { S7_SetPoint := 'True'} : Bool;   // Start dec. for reached requested position / Inizio dec. per raggiungimento quota richiesta
         xDecResearch { S7_SetPoint := 'True'} : Bool;   // Deceleration start for moving to level search speed / Inizio decelerazione per passaggio a velocità ricerca livello
         xStopVirPositioner { S7_SetPoint := 'True'} : Bool;   // Stop positioner for pos. reached / Arresto posizionatore Target raggiunto
         xEnableJog { S7_SetPoint := 'True'} : Bool;   // Jog movement in progress / JOG movimento in corso
         f_PositionTarget { S7_SetPoint := 'True'} : Real;   // Posizione Richiesta Target
         fVirPos { S7_SetPoint := 'True'} : Real;   // Pos. virtual encoder positioner (mm) / Posizione encoder Asse virtuale (mm)
         f_SpeedReqCalc { S7_SetPoint := 'True'} : Real;   // Velocità TARGET autocalcolata su spazio destinazione
         fVirSpeed { S7_SetPoint := 'True'} : Real;   // Virtual encoder speed positioner (mm/sec) / Velocità Asse virtuale (mm/sec) TRA-LOG-COS
         fVirSpeedLinear { S7_SetPoint := 'True'} : Real;   // Velocità Asse LINEARE
         fVirSpeedLog { S7_SetPoint := 'True'} : Real;   // Velocità Asse LOGARITMICA
         fVirSpeedCos { S7_SetPoint := 'True'} : Real;   // Velocità Asse COSENO
         fCmdVirSpeed { S7_SetPoint := 'True'} : Real;   // Virtual encoder current sp(mm/sec) / Velocità richiesta Asse (mm/sec)
         fCmdVirSpeedMemo { S7_SetPoint := 'True'} : Real;   // Memo Velocità richiesta Asse (mm/sec)
         fCmdVirAcc { S7_SetPoint := 'True'} : Real;   // Acc requested for positioner (mm/sec^2) / Acc. richiesta Asse (mm/sec^2)
         fCmdVirDec { S7_SetPoint := 'True'} : Real;   // Dec. requested for positioner (mm/sec^2) / Dec. richiesta Asse (mm/sec^2)
         fLimVirDec { S7_SetPoint := 'True'} : Real;   // Max modulated dec. limit to stop / * Limite massimo dec. modulata per fermata
         fDecVirStop { S7_SetPoint := 'True'} : Real;   // Dec. requested for positioner stop height (mm/sec^2) / * Dec. richiesta per posizionatore stop quota (mm/sec^2)
         fCalcEncErr { S7_SetPoint := 'True'} : Real;   // Error between motor encoder current & real pos. (mm) / * Errore tra pos. attuale e reale encoder motore
         fJogSpeed { S7_SetPoint := 'True'} : Real;   // Speed gen. by jog movement (mm/sec) / Velocità JOG (mm/sec)
         fCmdJogSpeed { S7_SetPoint := 'True'} : Real;   // Speed request to jog movement (mm/sec) / Velocità richiesta JOG (mm/sec)
         fCmdJogAcc { S7_SetPoint := 'True'} : Real;   // Acc. requested for jog movement (mm/sec^2) / Acc. richiesta JOG (mm/sec^2)
         fCmdJogDec { S7_SetPoint := 'True'} : Real;   // Dec. requested for jog movement (mm/sec^2) / Dec. richiesta JOG (mm/sec^2)
         "fLim+Ppid" { S7_SetPoint := 'True'} : Real;   // Proportional action positive maximum limit (1/5 max speed) / Limite massimo positivo azione proporzionale (20% velocità massima)
         "fLim-Ppid" { S7_SetPoint := 'True'} : Real;   // Proportional action negative maximum limit (1/5 max speed) / Limite massimo negativo azione proporzionale (20% velocità massima)
         fCmdSpeedMot { S7_SetPoint := 'True'} : Real;   // Motor control speed from positioner o Jog / Velocità comando motore da POS o JOG
         fSuppCalcPpid { S7_SetPoint := 'True'} : Real;   // Proportional calculation supp. / App calcolo proporzionale
         fMemoMaxSpeed { S7_SetPoint := 'True'} : Real;   // Store maximum speed (mm/sec) / Memorizzo velocità massima (mm/sec)
         fPpid { S7_SetPoint := 'True'} : Real;   // Part P of Pid / Parte P del Pid
         fMemoOldPos { S7_SetPoint := 'True'} : Real;   // Quota Old/Position Old (mm)
         fAccOnWork { S7_SetPoint := 'True'} : Real;   // Accelerazione calcolata/imposta
         fDecOnWork { S7_SetPoint := 'True'} : Real;   // Decelerazione calcolata/imposta
         xTimBrakeDelay_Fwd : Bool;   // Ritardo sgancio freno FWD
         xTimBrakeDelay_Bkw : Bool;   // Ritardo sgancio freno BKW
         xTimStopEndPos : Bool;   // Ritardo allarme controllo fine posizionamento
         fCalc : Array[0..20] of Real;
         xCalc : Array[0..20] of Bool;
      END_STRUCT;
   END_VAR
   VAR
      TmrBrake_Fwd : IEC_TIMER;   // Timer sgancio freno FWD
      TmrBrake_Bkw : IEC_TIMER;   // Timer sgancio freno BKW
      Tmr_EndPos : IEC_TIMER;   // Timer allarme controllo fine posizionamento
      Tmr_DriveOnReq : IEC_TIMER;   // Timer OFF richiesta Drive Ready
      Tmr_OnMove : IEC_TIMER;
   END_VAR
   VAR_TEMP
      tfSuppCalc : Real;   // Calculation support / Appoggio per calcoli
      fSlopeAccLog : Real;
      fSlopeDecLog : Real;
      fSlopeAccCos : Real;
      fSlopeDecCos : Real;
      fCalcSpeed : Real;
      oxCmdMotorFWD : Bool;
      oxCmdMotorBKW : Bool;
      fCalcSpaceOff : Real;
      xDummy : Bool;
   END_VAR
   VAR CONSTANT
      PiGrego : Real := 3.141593;
      "100Sec" : Time := T#100s;
   END_VAR
   VAR_TEMP   // added for the SCL form of the ladder/FBD networks
      _w1 : Bool;
      _w2 : Bool;
      _w3 : Bool;
   END_VAR
BEGIN

REGION Network 1 (SCL): Autocalcolo velocità su spazio da percorrere
   IF #DataIn.xAutoSpeedDetect THEN
       IF #Cfg."xmm/degree" THEN
           IF ABS(#DataIn.ifPositionRequest - #DataIn.ifEncoder) >= #Cfg.fMaxSpeed / 2 THEN
               #Work.f_SpeedReqCalc := #DataIn.ifSpeedRequest;
           ELSE
               #fCalcSpeed := ABS(#DataIn.ifPositionRequest - #DataIn.ifEncoder);
               IF NOT #DataOut.oxCmdMotorForw AND NOT #DataOut.oxCmdMotorBack THEN
                   IF #fCalcSpeed <= #DataIn.ifSpeedRequest THEN
                       #Work.f_SpeedReqCalc := #fCalcSpeed;
                   ELSE
                       #Work.f_SpeedReqCalc := #DataIn.ifSpeedRequest;
                   END_IF;
               END_IF;
           END_IF;
       ELSE
           IF ABS(#DataIn.ifPositionRequest - #DataIn.ifEncoder) >= 60.0 THEN
               #Work.f_SpeedReqCalc := #DataIn.ifSpeedRequest;
           ELSE
               #fCalcSpeed := ABS(#DataIn.ifPositionRequest - #DataIn.ifEncoder);
               IF NOT #DataOut.oxCmdMotorForw AND NOT #DataOut.oxCmdMotorBack THEN
                   IF #fCalcSpeed <= #DataIn.ifSpeedRequest THEN
                       #Work.f_SpeedReqCalc := #fCalcSpeed;
                   ELSE
                       #Work.f_SpeedReqCalc := #DataIn.ifSpeedRequest;
                   END_IF;
               END_IF;
           END_IF;
       END_IF;
   ELSE
       #Work.f_SpeedReqCalc := #DataIn.ifSpeedRequest;
   END_IF;

   IF #Work.f_SpeedReqCalc > #Cfg.fMaxSpeed THEN
       #Work.f_SpeedReqCalc := #Cfg.fMaxSpeed;
   END_IF;
END_REGION

REGION Network 2: Memo Posizionatore abilitato per inversione
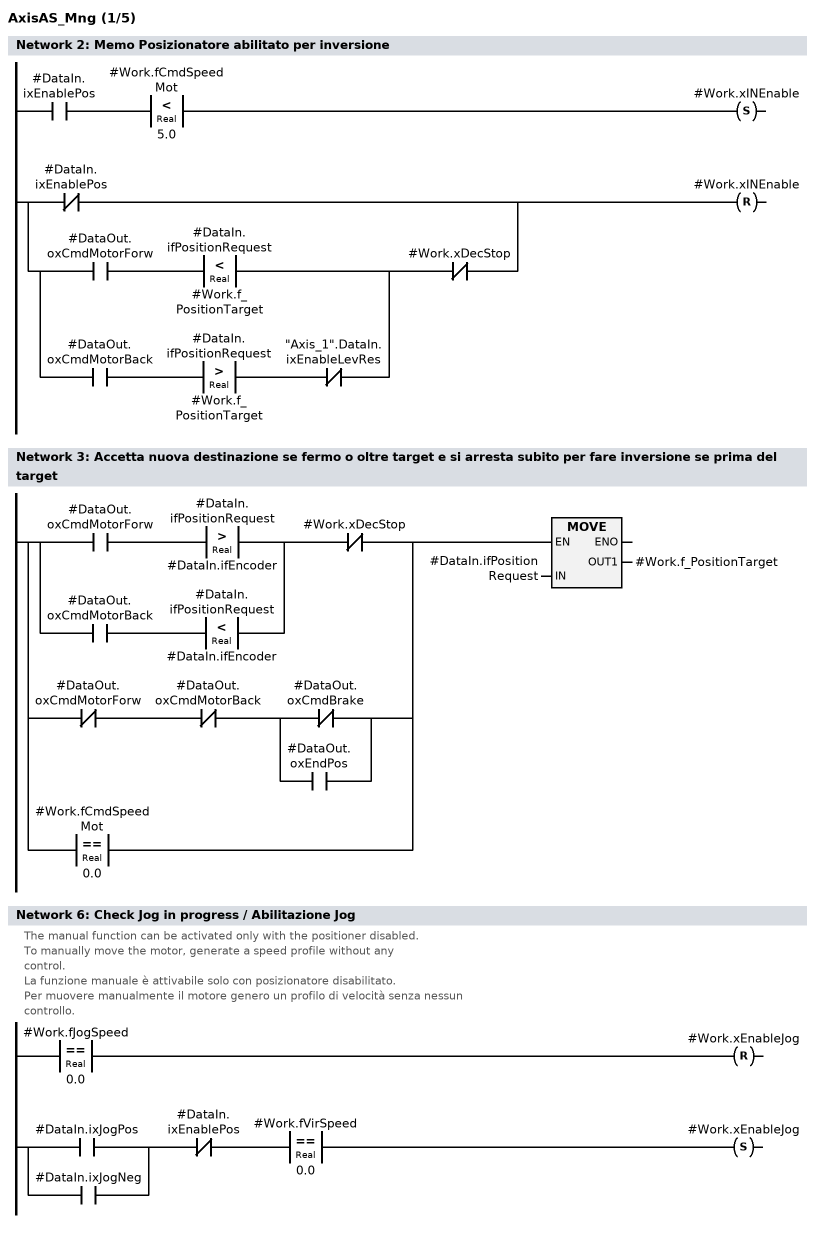
   RUNG wire#powerrail
      Contact( #DataIn.ixEnablePos )
      { S7_Templates := "SrcType := Real" } LT_Contact(in1 := #Work.fCmdSpeedMot, in2 := 5.0)
      S_Coil( #Work.xINEnable )
   END_RUNG
   RUNG wire#powerrail
      I_Contact( #DataIn.ixEnablePos )
      wire#w1
      R_Coil( #Work.xINEnable )
   END_RUNG
   RUNG wire#powerrail
      Contact( #DataOut.oxCmdMotorForw )
      { S7_Templates := "SrcType := Real" } LT_Contact(in1 := #DataIn.ifPositionRequest, in2 := #Work.f_PositionTarget)
      wire#w2
      I_Contact( #Work.xDecStop )
   END_RUNG wire#w1
   RUNG wire#powerrail
      Contact( #DataOut.oxCmdMotorBack )
      { S7_Templates := "SrcType := Real" } GT_Contact(in1 := #DataIn.ifPositionRequest, in2 := #Work.f_PositionTarget)
      I_Contact( "Axis_1".DataIn.ixEnableLevRes )
   END_RUNG wire#w2
   // the same network as SCL:
   IF #DataIn.ixEnablePos AND (#Work.fCmdSpeedMot < 5.0) THEN #Work.xINEnable := TRUE; END_IF;
   IF NOT #DataIn.ixEnablePos OR (((#DataOut.oxCmdMotorForw AND (#DataIn.ifPositionRequest < #Work.f_PositionTarget)) OR (#DataOut.oxCmdMotorBack AND (#DataIn.ifPositionRequest > #Work.f_PositionTarget) AND NOT "Axis_1".DataIn.ixEnableLevRes)) AND NOT #Work.xDecStop) THEN
       #Work.xINEnable := FALSE;
   END_IF;
END_REGION

REGION Network 3: Accetta nuova destinazione se fermo o oltre target e si arresta subito per fare inversione se prima del target
   RUNG wire#powerrail
      Contact( #DataOut.oxCmdMotorForw )
      { S7_Templates := "SrcType := Real" } GT_Contact(in1 := #DataIn.ifPositionRequest, in2 := #DataIn.ifEncoder)
      wire#w1
      I_Contact( #Work.xDecStop )
      wire#w2
      Move(in := #DataIn.ifPositionRequest, out1 => #Work.f_PositionTarget)
   END_RUNG
   RUNG wire#powerrail
      Contact( #DataOut.oxCmdMotorBack )
      { S7_Templates := "SrcType := Real" } LT_Contact(in1 := #DataIn.ifPositionRequest, in2 := #DataIn.ifEncoder)
   END_RUNG wire#w1
   RUNG wire#powerrail
      I_Contact( #DataOut.oxCmdMotorForw )
      I_Contact( #DataOut.oxCmdMotorBack )
      wire#w3
      I_Contact( #DataOut.oxCmdBrake )
   END_RUNG wire#w2
   RUNG wire#w3
      Contact( #DataOut.oxEndPos )
   END_RUNG wire#w2
   RUNG wire#powerrail
      { S7_Templates := "SrcType := Real" } EQ_Contact(in1 := #Work.fCmdSpeedMot, in2 := 0.0)
   END_RUNG wire#w2
   // the same network as SCL:
   IF (((#DataOut.oxCmdMotorForw AND (#DataIn.ifPositionRequest > #DataIn.ifEncoder)) OR (#DataOut.oxCmdMotorBack AND (#DataIn.ifPositionRequest < #DataIn.ifEncoder))) AND NOT #Work.xDecStop) OR (NOT #DataOut.oxCmdMotorForw AND NOT #DataOut.oxCmdMotorBack AND (NOT #DataOut.oxCmdBrake OR #DataOut.oxEndPos)) OR (#Work.fCmdSpeedMot = 0.0) THEN
       #Work.f_PositionTarget := #DataIn.ifPositionRequest;
   END_IF;
END_REGION

REGION Network 4 (SCL): Autocalcolo ACC-DEC su velocità
   IF #DataIn.xAutoAccDecCalculation THEN

       #Work.fAccOnWork := #Cfg.fMaxAccRamp * (#Work.f_SpeedReqCalc / #Cfg.fMaxSpeed);
       #Work.fDecOnWork := #Cfg.fMaxDecRamp * (#Work.f_SpeedReqCalc / #Cfg.fMaxSpeed);

       IF #Cfg."xmm/degree" THEN
           IF #Work.fAccOnWork < 100 THEN
               #Work.fAccOnWork := 100;
           END_IF;
           IF #Work.fDecOnWork < 100 THEN
               #Work.fDecOnWork := 100;
           END_IF;
       ELSE
           IF #Work.fAccOnWork < 20 THEN
               #Work.fAccOnWork := 20;
           END_IF;
           IF #Work.fDecOnWork < 20 THEN
               #Work.fDecOnWork := 20;
           END_IF;
       END_IF;

   ELSE

       #Work.fAccOnWork := #DataIn.ifAccRamp;
       #Work.fDecOnWork := #DataIn.ifDecRamp;

   END_IF;
END_REGION

REGION Network 5 (SCL): Encoder value conversion / Selezione curva
   // Per spostamenti inferiori a  #CFG."fAutoChangeS-Lvalue" impone una curva a TRA se selezionata LOG
   IF #Cfg."xCurveS-L" = 0 THEN
       #Work."xCurveS-L" := FALSE;
   END_IF;

   IF #Cfg."xCurveS-L" = 1 THEN
       IF (#Work.xINEnable) AND NOT #Work."xCTRAutoChangeS-L" THEN
           #Work."xCTRAutoChangeS-L" := TRUE;
           IF (ABS(#Work.f_PositionTarget - #DataOut.ofEncMotorPos) < #Cfg."fAutoChangeS-Lvalue") THEN
               #Work."xAutoChangeS-L" := TRUE;
           END_IF;
       END_IF;
       IF #Work."xAutoChangeS-L" THEN
           #Work."xCurveS-L" := FALSE;
       ELSE
           #Work."xCurveS-L" := TRUE;
       END_IF;
   END_IF;

   IF #Cfg."xCurveS-L" = 2 THEN
       #Work."xCurveS-L" := TRUE;
   END_IF;

   IF NOT #Work.xINEnable AND NOT #Work.xDecStop THEN
       #Work."xCTRAutoChangeS-L" := FALSE;
   END_IF;

   IF ABS(#Work.f_PositionTarget - #DataOut.ofEncMotorPos) <= #Cfg.fVirt_EncWindPos THEN
       #Work."xAutoChangeS-L" := FALSE;

   END_IF;
END_REGION

REGION Network 6: Check Jog in progress / Abilitazione Jog
   // The manual function can be activated only with the positioner disabled.
   // To manually move the motor, generate a speed profile without any 
   // control.
   // La funzione manuale è attivabile solo con posizionatore disabilitato.
   // Per muovere manualmente il motore genero un profilo di velocità senza nessun 
   // controllo.
   RUNG wire#powerrail
      { S7_Templates := "SrcType := Real" } EQ_Contact(in1 := #Work.fJogSpeed, in2 := 0.0)
      R_Coil( #Work.xEnableJog )
   END_RUNG
   RUNG wire#powerrail
      Contact( #DataIn.ixJogPos )
      wire#w1
      I_Contact( #DataIn.ixEnablePos )
      { S7_Templates := "SrcType := Real" } EQ_Contact(in1 := #Work.fVirSpeed, in2 := 0.0)
      S_Coil( #Work.xEnableJog )
   END_RUNG
   RUNG wire#powerrail
      Contact( #DataIn.ixJogNeg )
   END_RUNG wire#w1
   // the same network as SCL:
   IF #Work.fJogSpeed = 0.0 THEN #Work.xEnableJog := FALSE; END_IF;
   IF (#DataIn.ixJogPos OR #DataIn.ixJogNeg) AND NOT #DataIn.ixEnablePos AND (#Work.fVirSpeed = 0.0) THEN
       #Work.xEnableJog := TRUE;
   END_IF;
END_REGION

REGION Network 7 (SCL): Jog operation activation / Attivazione funzionamento di jog
   // Con abilitazione attiva carico velocità jog e inizio generazione profilo di velocità senza alcun controllo
   IF #Work.xEnableJog THEN

       IF #DataIn.ixJogPos OR #DataIn.ixJogNeg THEN
           #Work.fCmdJogSpeed := #Cfg.fJogSpeed;
       ELSE
           #Work.fCmdJogSpeed := 0.0;
       END_IF;

       IF #Work.fJogSpeed >= 0.0 THEN
           #Work.fCmdJogAcc := #Cfg.fJogAcc * #DataIn.ifTimeScan;
           #Work.fCmdJogDec := #Cfg.fJogDec * #DataIn.ifTimeScan;
       END_IF;

       IF #Work.fCmdJogSpeed > #Work.fJogSpeed THEN
           #Work.fJogSpeed := #Work.fJogSpeed + #Work.fCmdJogAcc;
           IF #Work.fJogSpeed > #Work.fCmdJogSpeed THEN
               #Work.fJogSpeed := #Work.fCmdJogSpeed;
           END_IF;
       END_IF;

       IF #Work.fCmdJogSpeed < #Work.fJogSpeed THEN
           #Work.fJogSpeed := #Work.fJogSpeed - #Work.fCmdJogDec;
           IF #Work.fJogSpeed < #Work.fCmdJogSpeed THEN
               #Work.fJogSpeed := #Work.fCmdJogSpeed;
           END_IF;
       END_IF;

   END_IF;
END_REGION

REGION Network 8: Check if positioner is enabled / Controllo se posizionatore abilitato e inverter ready
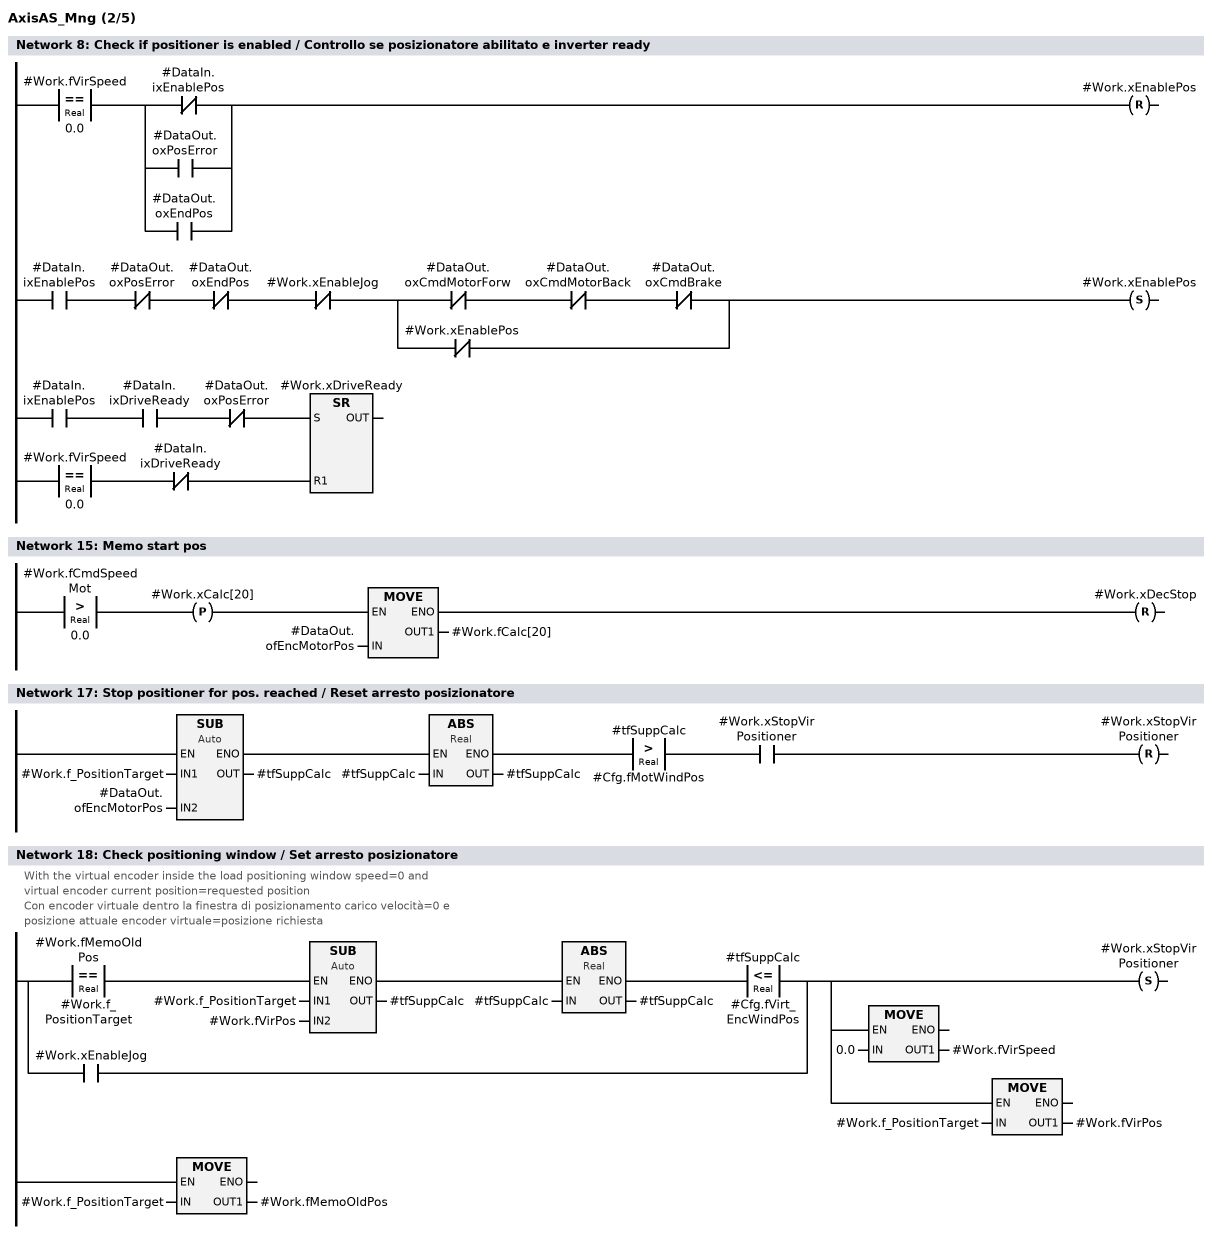
   RUNG wire#powerrail
      { S7_Templates := "SrcType := Real" } EQ_Contact(in1 := #Work.fVirSpeed, in2 := 0.0)
      wire#w1
      I_Contact( #DataIn.ixEnablePos )
      wire#w2
      R_Coil( #Work.xEnablePos )
   END_RUNG
   RUNG wire#w1
      Contact( #DataOut.oxPosError )
   END_RUNG wire#w2
   RUNG wire#w1
      Contact( #DataOut.oxEndPos )
   END_RUNG wire#w2
   RUNG wire#powerrail
      Contact( #DataIn.ixEnablePos )
      I_Contact( #DataOut.oxPosError )
      I_Contact( #DataOut.oxEndPos )
      I_Contact( #Work.xEnableJog )
      wire#w3
      I_Contact( #DataOut.oxCmdMotorForw )
      I_Contact( #DataOut.oxCmdMotorBack )
      I_Contact( #DataOut.oxCmdBrake )
      wire#w4
      S_Coil( #Work.xEnablePos )
   END_RUNG
   RUNG wire#w3
      I_Contact( #Work.xEnablePos )
   END_RUNG wire#w4
   RUNG wire#powerrail
      Contact( #DataIn.ixEnablePos )
      Contact( #DataIn.ixDriveReady )
      I_Contact( #DataOut.oxPosError )
      S_SR(operand := #Work.xDriveReady, r1 := wire#w5)
   END_RUNG
   RUNG wire#powerrail
      { S7_Templates := "SrcType := Real" } EQ_Contact(in1 := #Work.fVirSpeed, in2 := 0.0)
      I_Contact( #DataIn.ixDriveReady )
   END_RUNG wire#w5
   // the same network as SCL:
   IF (#Work.fVirSpeed = 0.0) AND (NOT #DataIn.ixEnablePos OR #DataOut.oxPosError OR #DataOut.oxEndPos) THEN
       #Work.xEnablePos := FALSE;
   END_IF;
   IF #DataIn.ixEnablePos AND NOT #DataOut.oxPosError AND NOT #DataOut.oxEndPos AND NOT #Work.xEnableJog AND ((NOT #DataOut.oxCmdMotorForw AND NOT #DataOut.oxCmdMotorBack AND NOT #DataOut.oxCmdBrake) OR NOT #Work.xEnablePos) THEN
       #Work.xEnablePos := TRUE;
   END_IF;
   IF #DataIn.ixEnablePos AND #DataIn.ixDriveReady AND NOT #DataOut.oxPosError THEN
       #Work.xDriveReady := TRUE;   // SR flip-flop
   END_IF;
   IF (#Work.fVirSpeed = 0.0) AND NOT #DataIn.ixDriveReady THEN #Work.xDriveReady := FALSE; END_IF;
END_REGION

REGION Network 9 (SCL): Calcolo Profilo velocità posizionatore TRAPEZIO

   #Work.fCmdVirAcc := (#Work.fAccOnWork * #DataIn.ifTimeScan);
   #Work.fCmdVirDec := (#Work.fDecOnWork * #DataIn.ifTimeScan);

   IF #Work.fCmdVirSpeed > #Work.fVirSpeedLinear THEN
       #Work.fVirSpeedLinear := #Work.fVirSpeedLinear + #Work.fCmdVirAcc;
       IF #Work.fVirSpeedLinear > #Work.fCmdVirSpeed THEN
           #Work.fVirSpeedLinear := #Work.fCmdVirSpeed;
       END_IF;
   END_IF;

   IF #Work.fCmdVirSpeed <= #Work.fVirSpeedLinear THEN
       #Work.fVirSpeedLinear := #Work.fVirSpeedLinear - #Work.fCmdVirDec;
       IF #Work.fVirSpeedLinear < #Work.fCmdVirSpeed THEN
           #Work.fVirSpeedLinear := #Work.fCmdVirSpeed;
       END_IF;
       IF NOT (#Work.xStopVirPositioner) AND (#Work.fVirSpeedLinear < #Cfg.fMinSpeed)
           AND NOT (#DataOut.oxPosError) AND #Work.xINEnable AND #Work.xDriveReady THEN
           #Work.fVirSpeedLinear := #Cfg.fMinSpeed;
       END_IF;
   END_IF;
END_REGION

REGION Network 10 (SCL): Gestione cambio target velocità LOG-COS
       IF (#Work.fCmdVirSpeedMemo <> #Work.fCmdVirSpeed) THEN
           IF #Work.fCmdVirSpeed > 0 AND #Work.fCmdVirSpeedMemo <> 0 THEN
               #Work.fCalc[7] := #Work.fVirSpeedLog;
               #Work.fCalc[0] := 0;
               #Work.fCalc[17] := #Work.fVirSpeedCos;
               #Work.fCalc[19] := 0;
               IF #Work.fCmdVirSpeed > #Work.fCmdVirSpeedMemo THEN
                   #Work.xCmdVirSpeedChanged := FALSE;
               ELSE
                   #Work.xCmdVirSpeedChanged := TRUE;
               END_IF;
           END_IF;
           #Work.fCmdVirSpeedMemo := #Work.fCmdVirSpeed;
       END_IF;
END_REGION

REGION Network 11 (SCL): Calculate positioner speed / Calcolo Profilo velocità posizionatore Logaritmica
   // Calculate speed positioner profile.
   // During the stop phase, module the deceleration to stop in the position 
   // requested; the maximum deceleration variation is 50%. This is 
   // necessary because the 0 speed request point is afflicted by an error 
   // generated by the CPU scanning time.
   // Calcolo velocità profilo posizionatore.
   // Durante la fase di fermata modulo la decelerazione per fermarmi nella posizione 
   // richiesta; la variazione massima di decelerazione è del 50%. Questo è 
   // necessario in quanto il punto di richiesta velocità 0 è afflitto dall'errore 
   // generato dal tempo di scansione della CPU.

   IF #Work."xCurveS-L" THEN



       IF  #Work.fCalc[10] < #Work.fVirSpeedLog THEN
           #Work.fCalc[10] := #Work.fVirSpeedLog;
       END_IF;
       IF #Work.fVirSpeed = 0 THEN
           #Work.fCalc[10] := 0;
       END_IF;


       #fSlopeAccLog := (12 * #Work.fAccOnWork) / (ABS(#Work.fCmdVirSpeed - #Work.fCalc[7]) + 1);
       #fSlopeDecLog := (12 * #Work.fDecOnWork) / (#Work.fCalc[10] + 1);


       IF #Work.fCmdVirSpeed > 0 THEN

           #Work.fCalc[5] := 1;
           IF #Work.fCalc[5] < #Work.fVirSpeedLog THEN
               #Work.fCalc[5] := #Work.fVirSpeedLog;
           END_IF;
           #Work.fCalc[0] := #Work.fCalc[0] + #DataIn.ifTimeScan;
           IF NOT #Work.xCmdVirSpeedChanged THEN
               #Work.fVirSpeedLog := #Work.fCalc[7] + (#Work.fCmdVirSpeed - #Work.fCalc[7]) * (1 / (1 + EXP(- (#Work.fCalc[0] * #fSlopeAccLog - #Cfg.fFirstStepNepero))));
           ELSE
               #fSlopeDecLog := (12 * #Work.fDecOnWork) / ABS((#Work.fCalc[7] - #Work.fCmdVirSpeed) + 1);
               #Work.fVirSpeedLog := #Work.fCalc[7] + (#Work.fCmdVirSpeed - #Work.fCalc[7]) * (1 / (1 + EXP(- (#Work.fCalc[0] * #fSlopeDecLog - #Cfg.fFirstStepNepero))));
           END_IF;

           #Work.fCalc[4] := 0;


       ELSE

           IF #Work.fVirSpeedLog > 0 THEN
               #Work.fCalc[4] := #Work.fCalc[4] + #DataIn.ifTimeScan;
           END_IF;
           #fSlopeDecLog := (12 * #Work.fDecOnWork) / (#Work.fCalc[5] + 1);
           #Work.fVirSpeedLog := #Work.fCalc[5] * (1 - (1 / (1 + EXP(- ((#Work.fCalc[4]) * #fSlopeDecLog - #Cfg.fFirstStepNepero)))));
           #Work.fCalc[10] := #Work.fCalc[5];
           #Work.fCalc[7] := #Work.fVirSpeedLog;
           #Work.fCalc[0] := 0;
       END_IF;


       IF #Work.xStopVirPositioner THEN
               #Work.fVirSpeed := 0;
               #Work.fCalc[0] := 0;
               #Work.fCalc[4] := 0;
               #Work.fCalc[5] := 0;
               #Work.fCalc[7] := 0;
        END_IF;

   END_IF;
END_REGION

REGION Network 12 (SCL): Calculate positioner speed / Calcolo Profilo velocità posizionatore Coseno
   // Calculate speed positioner profile.
   // During the stop phase, module the deceleration to stop in the position 
   // requested; the maximum deceleration variation is 50%. This is 
   // necessary because the 0 speed request point is afflicted by an error 
   // generated by the CPU scanning time.
   // Calcolo velocità profilo posizionatore.
   // Durante la fase di fermata modulo la decelerazione per fermarmi nella posizione 
   // richiesta; la variazione massima di decelerazione è del 50%. Questo è 
   // necessario in quanto il punto di richiesta velocità 0 è afflitto dall'errore 
   // generato dal tempo di scansione della CPU.

   IF #Work."xCurveS-L" THEN


       IF #Work.fCmdVirSpeed > 0 THEN

           #Work.fCalc[19] := #Work.fCalc[19] + #DataIn.ifTimeScan;

                   #Work.fCalc[13] := 1;
                   IF #Work.fCalc[13] < #Work.fVirSpeedCos THEN
                       #Work.fCalc[13] := #Work.fVirSpeedCos;
                   END_IF;
                   #fSlopeAccCos := #PiGrego / ((ABS(#Work.fCmdVirSpeed - #Work.fCalc[17]) + 1) / #Work.fAccOnWork);
                   IF NOT #Work.xCmdVirSpeedChanged THEN
                       IF #fSlopeAccCos * #Work.fCalc[19] < #PiGrego THEN
                           #Work.fVirSpeedCos := #Work.fCalc[17] + (#Work.fCmdVirSpeed - #Work.fCalc[17]) * 0.5 * (COS(#fSlopeAccCos * #Work.fCalc[19] + #PiGrego) + 1);
                       ELSE
                           #Work.fVirSpeedCos := #Work.fCmdVirSpeed;
                       END_IF;
                   ELSE
                       #fSlopeDecCos := #PiGrego / ((ABS(#Work.fCmdVirSpeed - #Work.fCalc[17]) + 1) / #Work.fDecOnWork);
                       IF #fSlopeDecCos * #Work.fCalc[19] < #PiGrego THEN
                           #Work.fVirSpeedCos := #Work.fCalc[17] + (#Work.fCmdVirSpeed - #Work.fCalc[17]) * 0.5 * (COS(#fSlopeDecCos * #Work.fCalc[19] + #PiGrego) + 1);
                       ELSE
                           #Work.fVirSpeedCos := #Work.fCmdVirSpeed;
                       END_IF;

                   END_IF;
               #Work.fCalc[18] := #DataIn.ifTimeScan * 0;

           ELSE
               #Work.fCalc[19] := 0;
               IF #Work.fVirSpeedCos > 0 THEN
                   #Work.fCalc[18] := #Work.fCalc[18] + #DataIn.ifTimeScan;
                   #fSlopeDecCos := #PiGrego / (#Work.fCalc[13] / #Work.fDecOnWork);
                   IF #fSlopeDecCos * #Work.fCalc[18] < #PiGrego THEN
                       #Work.fVirSpeedCos := #Work.fCalc[13] * 0.5 * (COS(#fSlopeDecCos * #Work.fCalc[18]) + 1);
                   ELSE
                       #Work.fVirSpeedCos := 0;
                   END_IF;
                   #Work.fCalc[17] := #Work.fVirSpeedCos;
                   #Work.fCalc[19] := 0;
               END_IF;


       END_IF;


           IF #Work.xStopVirPositioner THEN
               #Work.fVirSpeed := 0;
               #Work.fCalc[13] := 0;
               #Work.fCalc[17] := 0;
               #Work.fCalc[18] := 0;
               #Work.fCalc[19] := 0;
           END_IF;


   END_IF;
END_REGION

REGION Network 13 (SCL): Gestione profilo posizionatore

   IF NOT #Work.xStopVirPositioner THEN

       CASE #Cfg."xCurveS-L" OF
           0:
               #Work.fVirSpeed := #Work.fVirSpeedLinear;
           1:
               IF #Work."xCurveS-L" THEN
                   IF #Work.fVirSpeedLog >= 1 THEN
                       #Work.fVirSpeed := #Work.fVirSpeedLog;
                   ELSE
                       #Work.fVirSpeed := 0;
                   END_IF;
               ELSE
                   #Work.fVirSpeed := #Work.fVirSpeedLinear;
               END_IF;

           2:
               #Work.fVirSpeed := #Work.fVirSpeedCos;

       END_CASE;


       IF (#Work.fVirSpeed < #Cfg.fMinSpeed) AND #Work.xINEnable AND NOT (#DataOut.oxPosError) AND #Work.xDriveReady THEN
           #Work.fVirSpeed := #Cfg.fMinSpeed;
       END_IF;
   ELSE
       #Work.xCmdVirSpeedChanged := FALSE;
   END_IF;
END_REGION

REGION Network 14 (SCL): Calculate pos. compared to speed / Calcolo posizione con legge di moto
   // Calculate the profile generator position according to speed and time 
   // for scanning of the CPU.
   // The virtual encoder generated in this way is needed to calculate the PID managing the 
   // motor
   // Calcolo la posizione del generatore di profilo sul tempo 
   // di scansione della CPU.
   IF NOT #Work.xStopVirPositioner THEN
       IF #Work.f_PositionTarget > #Work.fVirPos THEN
           #Work.fVirPos := #Work.fVirPos + (#Work.fVirSpeed * #DataIn.ifTimeScan);
       ELSE
           #Work.fVirPos := #Work.fVirPos - (#Work.fVirSpeed * #DataIn.ifTimeScan);
       END_IF;
   END_IF;
END_REGION

REGION Network 15: Memo start pos
   RUNG wire#powerrail
      { S7_Templates := "SrcType := Real" } GT_Contact(in1 := #Work.fCmdSpeedMot, in2 := 0.0)
      P_Trig( #Work.xCalc[20] )
      Move(in := #DataOut.ofEncMotorPos, out1 => #Work.fCalc[20])
      R_Coil( #Work.xDecStop )
   END_RUNG
   // the same network as SCL:
   #_w1 := #Work.fCmdSpeedMot > 0.0;
   #_w2 := #_w1 AND NOT #Work.xCalc[20];   // rising edge
   #Work.xCalc[20] := #_w1;
   IF #_w2 THEN
       #Work.fCalc[20] := #DataOut.ofEncMotorPos;
       #Work.xDecStop := FALSE;
   END_IF;
END_REGION

REGION Network 16 (SCL): Check when it is time to bring the speed to 0 to stop / Calcolo spazio di arresto del profilo con dati attuali
   #DataOut.ofSpaceStop := #Cfg.fMotWindPos + #Cfg.fMotAdvStopPosition + (SQR(#Work.fVirSpeed)) / (#Work.fDecOnWork * 2.0);
   #DataOut.ofSpaceStart := (SQR(#Work.fCmdVirSpeed)) / (#Work.fAccOnWork * 2.0);
   #DataOut.ofSpaceLevRes := (SQR(#Work.fVirSpeed) / (#Work.fDecOnWork * 2.0)) - (SQR( #DataIn.ifSpeedLev) / (#Work.fDecOnWork * 2.0)) + 50;
   // #OUT.ofSpaceLevRes := (SQR(#WORK.f_SpeedReqCalc ) / (#IN.ifDecRamp * 2.0)) - (SQR( #IN.ifSpeedLev) / (#IN.ifDecRamp * 2.0));

   #DataOut.oxAccOnWork := ABS(#Work.fCalc[20] - #DataOut.ofEncMotorPos) < #DataOut.ofSpaceStart;
   #DataOut.oxDecOnWork := #Work.xDecStop OR ((#Work.fCmdSpeedMot > 0) AND NOT #Work.xINEnable);


   IF (ABS(#Work.f_PositionTarget - #Work.fVirPos)) <= #DataOut.ofSpaceStop THEN
       #Work.xDecStop := 1;
   END_IF;

   IF NOT (#Work.xEnablePos) OR #Work.xStopVirPositioner THEN //OR (NOT(#OUT.oxCmdMotorForw) AND NOT(#OUT.oxCmdMotorBack)) THEN
       #Work.xDecStop := 0;
   END_IF;


   IF #DataIn.ixEnableLevRes AND #Work.xINEnable THEN //AND (#SUPPORT.fVirSpeed > 0)   AND  #OUT.oxCmdMotorBack
       IF #DataIn.ifEncoder < (#DataIn.ifPositionStartLev + #DataOut.ofSpaceLevRes + 1) THEN
           #Work.xDecResearch := 1;
       END_IF;
   ELSE
       #Work.xDecResearch := 0;
   END_IF;
END_REGION

REGION Network 17: Stop positioner for pos. reached / Reset arresto posizionatore
   RUNG wire#powerrail
      Sub(in1 := #Work.f_PositionTarget, in2 := #DataOut.ofEncMotorPos, out => #tfSuppCalc)
      { S7_Templates := "SrcType := Real" } Abs(in := #tfSuppCalc, out => #tfSuppCalc)
      { S7_Templates := "SrcType := Real" } GT_Contact(in1 := #tfSuppCalc, in2 := #Cfg.fMotWindPos)
      Contact( #Work.xStopVirPositioner )
      R_Coil( #Work.xStopVirPositioner )
   END_RUNG
   // the same network as SCL:
   #tfSuppCalc := #Work.f_PositionTarget - #DataOut.ofEncMotorPos;
   #tfSuppCalc := ABS(#tfSuppCalc);
   IF (#tfSuppCalc > #Cfg.fMotWindPos) AND #Work.xStopVirPositioner THEN
       #Work.xStopVirPositioner := FALSE;
   END_IF;
END_REGION

REGION Network 18: Check positioning window / Set arresto posizionatore
   // With the virtual encoder inside the load positioning window speed=0 and 
   // virtual encoder current position=requested position
   // Con encoder virtuale dentro la finestra di posizionamento carico velocità=0 e 
   // posizione attuale encoder virtuale=posizione richiesta
   RUNG wire#powerrail
      { S7_Templates := "SrcType := Real" } EQ_Contact(in1 := #Work.fMemoOldPos, in2 := #Work.f_PositionTarget)
      Sub(in1 := #Work.f_PositionTarget, in2 := #Work.fVirPos, out => #tfSuppCalc)
      { S7_Templates := "SrcType := Real" } Abs(in := #tfSuppCalc, out => #tfSuppCalc)
      { S7_Templates := "SrcType := Real" } LE_Contact(in1 := #tfSuppCalc, in2 := #Cfg.fVirt_EncWindPos)
      wire#w1
      S_Coil( #Work.xStopVirPositioner )
   END_RUNG
   RUNG wire#powerrail
      Contact( #Work.xEnableJog )
   END_RUNG wire#w1
   RUNG wire#w1
      Move(in := 0.0, out1 => #Work.fVirSpeed)
   END_RUNG
   RUNG wire#w1
      Move(in := #Work.f_PositionTarget, out1 => #Work.fVirPos)
   END_RUNG
   RUNG wire#powerrail
      Move(in := #Work.f_PositionTarget, out1 => #Work.fMemoOldPos)
   END_RUNG
   // the same network as SCL:
   #_w1 := #Work.fMemoOldPos = #Work.f_PositionTarget;
   IF #_w1 THEN
       #tfSuppCalc := #Work.f_PositionTarget - #Work.fVirPos;
       #tfSuppCalc := ABS(#tfSuppCalc);
   END_IF;
   IF (#_w1 AND (#tfSuppCalc <= #Cfg.fVirt_EncWindPos)) OR #Work.xEnableJog THEN
       #Work.xStopVirPositioner := TRUE;
       #Work.fVirSpeed := 0.0;
       #Work.fVirPos := #Work.f_PositionTarget;
   END_IF;
   #Work.fMemoOldPos := #Work.f_PositionTarget;
END_REGION

REGION Network 19: Positioning speed requested / Velocità richiesta
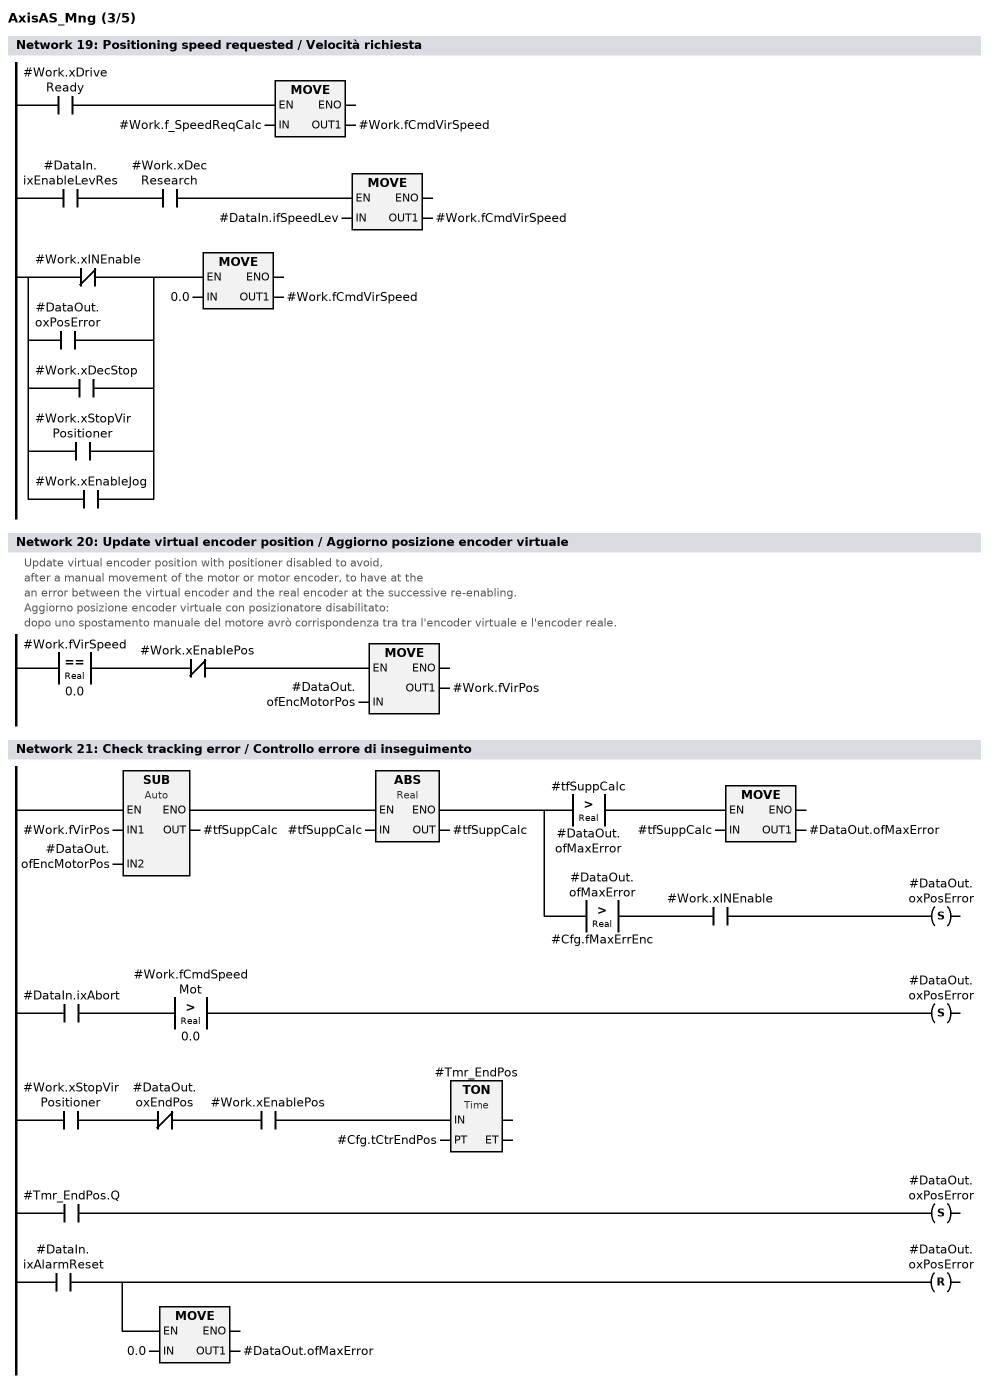
   RUNG wire#powerrail
      Contact( #Work.xDriveReady )
      Move(in := #Work.f_SpeedReqCalc, out1 => #Work.fCmdVirSpeed)
   END_RUNG
   RUNG wire#powerrail
      Contact( #DataIn.ixEnableLevRes )
      Contact( #Work.xDecResearch )
      Move(in := #DataIn.ifSpeedLev, out1 => #Work.fCmdVirSpeed)
   END_RUNG
   RUNG wire#powerrail
      I_Contact( #Work.xINEnable )
      wire#w1
      Move(in := 0.0, out1 => #Work.fCmdVirSpeed)
   END_RUNG
   RUNG wire#powerrail
      Contact( #DataOut.oxPosError )
   END_RUNG wire#w1
   RUNG wire#powerrail
      Contact( #Work.xDecStop )
   END_RUNG wire#w1
   RUNG wire#powerrail
      Contact( #Work.xStopVirPositioner )
   END_RUNG wire#w1
   RUNG wire#powerrail
      Contact( #Work.xEnableJog )
   END_RUNG wire#w1
   // the same network as SCL:
   IF #Work.xDriveReady THEN #Work.fCmdVirSpeed := #Work.f_SpeedReqCalc; END_IF;
   IF #DataIn.ixEnableLevRes AND #Work.xDecResearch THEN #Work.fCmdVirSpeed := #DataIn.ifSpeedLev; END_IF;
   IF NOT #Work.xINEnable OR #DataOut.oxPosError OR #Work.xDecStop OR #Work.xStopVirPositioner OR #Work.xEnableJog THEN
       #Work.fCmdVirSpeed := 0.0;
   END_IF;
END_REGION

REGION Network 20: Update virtual encoder position / Aggiorno posizione encoder virtuale
   // Update virtual encoder position with positioner disabled to avoid, 
   // after a manual movement of the motor or motor encoder, to have at the 
   // an error between the virtual encoder and the real encoder at the successive re-enabling.
   // Aggiorno posizione encoder virtuale con posizionatore disabilitato: 
   // dopo uno spostamento manuale del motore avrò corrispondenza tra tra l'encoder virtuale e l'encoder reale.
   RUNG wire#powerrail
      { S7_Templates := "SrcType := Real" } EQ_Contact(in1 := #Work.fVirSpeed, in2 := 0.0)
      I_Contact( #Work.xEnablePos )
      Move(in := #DataOut.ofEncMotorPos, out1 => #Work.fVirPos)
   END_RUNG
   // the same network as SCL:
   IF (#Work.fVirSpeed = 0.0) AND NOT #Work.xEnablePos THEN #Work.fVirPos := #DataOut.ofEncMotorPos; END_IF;
END_REGION

REGION Network 21: Check tracking error / Controllo errore di inseguimento
   RUNG wire#powerrail
      Sub(in1 := #Work.fVirPos, in2 := #DataOut.ofEncMotorPos, out => #tfSuppCalc)
      { S7_Templates := "SrcType := Real" } Abs(in := #tfSuppCalc, out => #tfSuppCalc)
      wire#w1
      { S7_Templates := "SrcType := Real" } GT_Contact(in1 := #tfSuppCalc, in2 := #DataOut.ofMaxError)
      Move(in := #tfSuppCalc, out1 => #DataOut.ofMaxError)
   END_RUNG
   RUNG wire#w1
      { S7_Templates := "SrcType := Real" } GT_Contact(in1 := #DataOut.ofMaxError, in2 := #Cfg.fMaxErrEnc)
      Contact( #Work.xINEnable )
      S_Coil( #DataOut.oxPosError )
   END_RUNG
   RUNG wire#powerrail
      Contact( #DataIn.ixAbort )
      { S7_Templates := "SrcType := Real" } GT_Contact(in1 := #Work.fCmdSpeedMot, in2 := 0.0)
      S_Coil( #DataOut.oxPosError )
   END_RUNG
   RUNG wire#powerrail
      Contact( #Work.xStopVirPositioner )
      I_Contact( #DataOut.oxEndPos )
      Contact( #Work.xEnablePos )
      { S7_Templates := "time_type := Time" } #Tmr_EndPos.TON(pt := #Cfg.tCtrEndPos, et =>)
   END_RUNG
   RUNG wire#powerrail
      Contact( #Tmr_EndPos.Q )
      S_Coil( #DataOut.oxPosError )
   END_RUNG
   RUNG wire#powerrail
      Contact( #DataIn.ixAlarmReset )
      wire#w2
      R_Coil( #DataOut.oxPosError )
   END_RUNG
   RUNG wire#w2
      Move(in := 0.0, out1 => #DataOut.ofMaxError)
   END_RUNG
   // the same network as SCL:
   #tfSuppCalc := #Work.fVirPos - #DataOut.ofEncMotorPos;
   #tfSuppCalc := ABS(#tfSuppCalc);
   IF #tfSuppCalc > #DataOut.ofMaxError THEN #DataOut.ofMaxError := #tfSuppCalc; END_IF;
   IF (#DataOut.ofMaxError > #Cfg.fMaxErrEnc) AND #Work.xINEnable THEN #DataOut.oxPosError := TRUE; END_IF;
   IF #DataIn.ixAbort AND (#Work.fCmdSpeedMot > 0.0) THEN #DataOut.oxPosError := TRUE; END_IF;
   #Tmr_EndPos.TON(IN := #Work.xStopVirPositioner AND NOT #DataOut.oxEndPos AND #Work.xEnablePos,
                   PT := #Cfg.tCtrEndPos);
   IF #Tmr_EndPos.Q THEN #DataOut.oxPosError := TRUE; END_IF;
   IF #DataIn.ixAlarmReset THEN
       #DataOut.oxPosError := FALSE;
       #DataOut.ofMaxError := 0.0;
   END_IF;
END_REGION

REGION Network 22 (SCL): Calcolo correzione PID

   #Work."fLim+Ppid" :=   (#Cfg.fMaxSpeed * 0.2);
   #Work."fLim-Ppid" := - (#Cfg.fMaxSpeed * 0.2);


   IF (#DataIn.ixEnableLevRes AND #Work.xDecResearch AND NOT #Work.xDecStop) OR #DataOut.oxEndPos THEN
       #Work.fMemoMaxSpeed := 1;
   END_IF;

   IF (ABS(#Work.fVirSpeed) > #Work.fMemoMaxSpeed) THEN
       #Work.fMemoMaxSpeed := #Work.fVirSpeed;
   END_IF;
   #Work.fSuppCalcPpid := ((#Work.fMemoMaxSpeed - #Work.fVirSpeed) / #Work.fMemoMaxSpeed) * #Cfg.fKPpidDec_Pos + #Cfg.fKPpid_Pos;
END_REGION

REGION Network 23 (SCL): Amplifico correzione PID a piramide su posizionamento
   #Work.fPpid := (#Work.fVirPos - #DataOut.ofEncMotorPos) * #Work.fSuppCalcPpid;
   IF #DataOut.oxCmdMotorBack THEN
       #Work.fPpid := - (#Work.fVirPos - #DataOut.ofEncMotorPos) * #Work.fSuppCalcPpid;
   END_IF;


   IF #Work.fPpid > #Work."fLim+Ppid" THEN
       #Work.fPpid := #Work."fLim+Ppid";
   END_IF;
   IF #Work.fPpid < #Work."fLim-Ppid" THEN
       #Work.fPpid := #Work."fLim-Ppid";
   END_IF;

   //Con posizionatore disabilitato azzero la parte proporzionale

   IF NOT #Work.xEnablePos OR #Work.xStopVirPositioner OR #DataOut.oxPosError THEN
       #Work.fPpid := 0;
   END_IF;

   // IF NOT #WORK.xEnablePos OR #WORK.xStopPositioner OR
   //     #WORK.fVirSpeed <= #CFG.fMinSpeed OR
   //     (NOT(#WORK.xINEnable) AND #WORK.fVirSpeed < 10) OR
   //     (ABS(#WORK.fNewPositionReq - #IN.ifEncoder) < #CFG.fMotWindPos) OR #OUT.oxPosError THEN
   //     #WORK.fPpid := 0;
   // END_IF;
END_REGION

